C07320=1109.351,336.589,-83.150,-177.426,10.830,149.506
C07321=1109.354,336.377,-83.120,-177.429,10.829,149.507
C07322=1109.357,336.166,-83.091,-177.431,10.827,149.507
C07323=1109.361,335.954,-83.061,-177.435,10.824,149.507
C07324=1109.364,335.707,-83.027,-177.437,10.823,149.507
C07325=1109.368,335.458,-82.992,-177.440,10.820,149.507
C07326=1109.373,335.211,-82.959,-177.443,10.817,149.508
C07327=1109.376,334.963,-82.924,-177.447,10.815,149.508
C07328=1109.380,334.715,-82.890,-177.450,10.812,149.508
C07329=1109.385,334.468,-82.856,-177.453,10.810,149.508
C07330=1109.388,334.220,-82.822,-177.456,10.807,149.508
C07331=1109.393,333.973,-82.787,-177.460,10.805,149.509
C07332=1109.396,333.725,-82.753,-177.463,10.802,149.509
C07333=1109.400,333.478,-82.719,-177.466,10.799,149.509
C07334=1109.404,333.229,-82.685,-177.469,10.798,149.509
C07335=1109.408,332.982,-82.651,-177.472,10.795,149.509
C07336=1109.412,332.735,-82.617,-177.475,10.793,149.509
C07337=1109.416,332.487,-82.582,-177.478,10.790,149.510
C07338=1109.419,332.240,-82.549,-177.481,10.788,149.510
C07339=1109.424,331.991,-82.514,-177.484,10.785,149.510
C07340=1109.428,331.744,-82.481,-177.488,10.782,149.510
C07341=1109.431,331.497,-82.447,-177.491,10.780,149.510
C07342=1109.435,331.249,-82.412,-177.494,10.777,149.511
C07343=1109.440,331.001,-82.379,-177.497,10.776,149.511
C07344=1109.443,330.754,-82.345,-177.500,10.773,149.511
C07345=1109.447,330.506,-82.310,-177.503,10.771,149.511
C07346=1109.451,330.258,-82.277,-177.506,10.768,149.511
C07347=1109.455,330.011,-82.243,-177.510,10.765,149.512
C07348=1109.459,329.762,-82.209,-177.513,10.763,149.512
C07349=1109.463,329.515,-82.175,-177.516,10.760,149.512
C07350=1109.467,329.268,-82.141,-177.519,10.758,149.512
C07351=1109.471,329.019,-82.108,-177.522,10.755,149.512
C07352=1109.475,328.772,-82.074,-177.525,10.752,149.512
C07353=1109.479,328.524,-82.040,-177.528,10.751,149.513
C07354=1109.483,328.276,-82.006,-177.531,10.748,149.513
C07355=1109.487,328.029,-81.973,-177.534,10.746,149.513
C07356=1109.491,327.782,-81.939,-177.538,10.743,149.513
C07357=1109.496,327.534,-81.905,-177.541,10.741,149.513
C07358=1109.499,327.286,-81.871,-177.544,10.738,149.514
C07359=1109.503,327.038,-81.838,-177.547,10.735,149.514
C07360=1109.507,326.791,-81.804,-177.550,10.733,149.514
C07361=1109.510,326.543,-81.770,-177.553,10.730,149.514
C07362=1109.514,326.295,-81.736,-177.557,10.728,149.514
C07363=1109.519,326.047,-81.703,-177.559,10.726,149.515
C07364=1109.523,325.800,-81.669,-177.562,10.723,149.515
C07365=1109.526,325.552,-81.635,-177.566,10.721,149.515
C07366=1109.531,325.304,-81.602,-177.569,10.718,149.515
C07367=1109.534,325.057,-81.568,-177.572,10.716,149.515
C07368=1109.538,324.809,-81.535,-177.575,10.713,149.515
C07369=1109.543,324.562,-81.502,-177.579,10.711,149.516
C07370=1109.546,324.314,-81.468,-177.581,10.708,149.516
C07371=1109.550,324.066,-81.434,-177.585,10.706,149.516
C07372=1109.554,323.854,-81.406,-177.587,10.704,149.516
C07373=1109.557,323.642,-81.377,-177.590,10.702,149.516
C07374=1109.561,323.430,-81.348,-177.593,10.699,149.516
C07375=1109.564,323.219,-81.320,-177.595,10.697,149.517
C07376=1109.567,323.006,-81.291,-177.598,10.695,149.517
C07377=1109.571,322.794,-81.263,-177.601,10.693,149.517
C07378=1109.575,322.582,-81.234,-177.603,10.691,149.517
C07379=1109.577,322.370,-81.205,-177.606,10.689,149.517
C07380=1109.581,322.122,-81.172,-177.609,10.687,149.517
C07381=1109.586,321.874,-81.139,-177.612,10.684,149.518
C07382=1109.589,321.627,-81.105,-177.615,10.681,149.518
C07383=1109.594,321.379,-81.072,-177.618,10.679,149.518
C07384=1109.597,321.131,-81.039,-177.621,10.676,149.518
C07385=1109.601,320.883,-81.005,-177.625,10.674,149.518
C07386=1109.605,320.635,-80.972,-177.628,10.671,149.518
C07387=1109.609,320.388,-80.939,-177.630,10.669,149.519
C07388=1109.614,320.140,-80.906,-177.634,10.667,149.519
C07389=1109.618,319.892,-80.873,-177.637,10.664,149.519
C07390=1109.621,319.645,-80.840,-177.640,10.662,149.519
C07391=1109.625,319.397,-80.807,-177.643,10.659,149.519
C07392=1109.629,319.149,-80.773,-177.646,10.656,149.520
C07393=1109.633,318.902,-80.740,-177.649,10.654,149.520
C07394=1109.637,318.654,-80.707,-177.652,10.651,149.520
C07395=1109.641,318.406,-80.674,-177.656,10.649,149.520
C07396=1109.645,318.158,-80.641,-177.658,10.647,149.520
C07397=1109.650,317.910,-80.608,-177.661,10.644,149.520
C07398=1109.653,317.663,-80.575,-177.665,10.642,149.521
C07399=1109.657,317.415,-80.542,-177.668,10.639,149.521
C07400=1109.661,317.167,-80.509,-177.671,10.637,149.521
C07401=1109.665,316.919,-80.476,-177.674,10.634,149.521
C07402=1109.669,316.672,-80.443,-177.677,10.631,149.521
C07403=1109.672,316.424,-80.410,-177.681,10.629,149.522
C07404=1109.676,316.176,-80.377,-177.683,10.626,149.522
C07405=1109.681,315.928,-80.343,-177.687,10.624,149.522
C07406=1109.685,315.680,-80.311,-177.689,10.622,149.522
C07407=1109.689,315.432,-80.278,-177.692,10.619,149.522
C07408=1109.693,315.185,-80.245,-177.696,10.617,149.523
C07409=1109.697,314.937,-80.212,-177.699,10.614,149.523
C07410=1109.701,314.689,-80.179,-177.702,10.612,149.523
C07411=1109.705,314.441,-80.146,-177.705,10.609,149.523
C07412=1109.709,314.193,-80.114,-177.708,10.606,149.523
C07413=1109.713,313.946,-80.081,-177.711,10.604,149.523
C07414=1109.717,313.697,-80.048,-177.714,10.601,149.524
C07415=1109.721,313.450,-80.016,-177.717,10.600,149.524
C07416=1109.725,313.202,-79.983,-177.720,10.597,149.524
C07417=1109.729,312.954,-79.950,-177.723,10.594,149.524
C07418=1109.733,312.706,-79.918,-177.726,10.592,149.524
C07419=1109.737,312.459,-79.884,-177.730,10.589,149.524
C07420=1109.741,312.210,-79.852,-177.733,10.586,149.525
C07421=1109.745,311.964,-79.820,-177.736,10.584,149.525
C07422=1109.749,311.716,-79.787,-177.739,10.581,149.525
C07423=1109.754,311.468,-79.754,-177.742,10.579,149.525
C07424=1109.757,311.220,-79.722,-177.746,10.576,149.525
C07425=1109.762,310.972,-79.689,-177.748,10.574,149.525
C07426=1109.766,310.724,-79.656,-177.751,10.572,149.526
C07427=1109.769,310.476,-79.624,-177.754,10.569,149.526
C07428=1109.773,310.264,-79.596,-177.757,10.567,149.526
C07429=1109.776,310.052,-79.568,-177.760,10.565,149.526
C07430=1109.780,309.840,-79.540,-177.762,10.563,149.526
C07431=1109.783,309.627,-79.513,-177.765,10.560,149.527
C07432=1109.787,309.415,-79.484,-177.768,10.558,149.527
C07433=1109.790,309.203,-79.456,-177.770,10.556,149.527
C07434=1109.794,308.991,-79.429,-177.773,10.554,149.527
C07435=1109.797,308.779,-79.401,-177.776,10.552,149.527
C07436=1109.801,308.532,-79.369,-177.779,10.549,149.527
C07437=1109.805,308.283,-79.336,-177.782,10.546,149.527
C07438=1109.809,308.035,-79.304,-177.785,10.544,149.528
C07439=1109.814,307.788,-79.272,-177.787,10.542,149.528
C07440=1109.817,307.540,-79.240,-177.791,10.540,149.528
C07441=1109.822,307.292,-79.207,-177.794,10.537,149.528
C07442=1109.825,307.044,-79.175,-177.797,10.534,149.528
C07443=1109.830,306.796,-79.142,-177.800,10.532,149.528
C07444=1109.833,306.548,-79.111,-177.803,10.529,149.529
C07445=1109.838,306.301,-79.078,-177.806,10.526,149.529
C07446=1109.842,306.053,-79.046,-177.810,10.524,149.529
C07447=1109.846,305.804,-79.013,-177.812,10.521,149.529
C07448=1109.850,305.556,-78.982,-177.815,10.520,149.529
C07449=1109.854,305.309,-78.948,-177.818,10.517,149.529
C07450=1109.858,305.061,-78.917,-177.821,10.514,149.530
C07451=1109.862,304.813,-78.885,-177.824,10.512,149.530
C07452=1109.866,304.565,-78.853,-177.828,10.509,149.530
C07453=1109.870,304.317,-78.821,-177.831,10.506,149.530
C07454=1109.874,304.069,-78.788,-177.834,10.504,149.530
C07455=1109.879,303.822,-78.756,-177.837,10.502,149.531
C07456=1109.882,303.574,-78.724,-177.840,10.499,149.531
C07457=1109.887,303.325,-78.692,-177.843,10.497,149.531
C07458=1109.890,303.077,-78.660,-177.846,10.494,149.531
C07459=1109.895,302.830,-78.629,-177.849,10.492,149.531
C07460=1109.899,302.582,-78.596,-177.852,10.489,149.531
C07461=1109.903,302.334,-78.564,-177.855,10.487,149.532
C07462=1109.907,302.086,-78.533,-177.858,10.484,149.532
C07463=1109.912,301.838,-78.500,-177.862,10.482,149.532
C07464=1109.915,301.590,-78.469,-177.865,10.479,149.532
C07465=1109.919,301.342,-78.437,-177.868,10.476,149.532
C07466=1109.924,301.094,-78.405,-177.871,10.474,149.532
C07467=1109.928,300.846,-78.373,-177.874,10.472,149.533
C07468=1109.932,300.598,-78.341,-177.876,10.469,149.533
C07469=1109.936,300.351,-78.309,-177.880,10.467,149.533
C07470=1109.940,300.103,-78.277,-177.883,10.464,149.533
C07471=1109.944,299.854,-78.245,-177.886,10.461,149.533
C07472=1109.948,299.607,-78.214,-177.889,10.459,149.534
C07473=1109.952,299.359,-78.182,-177.892,10.456,149.534
C07474=1109.956,299.111,-78.150,-177.895,10.454,149.534
C07475=1109.961,298.863,-78.118,-177.899,10.451,149.534
C07476=1109.964,298.615,-78.086,-177.901,10.449,149.534
C07477=1109.968,298.367,-78.054,-177.904,10.447,149.535
C07478=1109.973,298.119,-78.023,-177.907,10.444,149.535
C07479=1109.976,297.871,-77.992,-177.910,10.441,149.535
C07480=1109.980,297.623,-77.960,-177.913,10.439,149.535
C07481=1109.985,297.376,-77.928,-177.916,10.436,149.535
C07482=1109.989,297.128,-77.896,-177.920,10.433,149.535
C07483=1109.993,296.879,-77.865,-177.923,10.431,149.535
C07484=1109.997,296.667,-77.838,-177.925,10.429,149.536
C07485=1110.000,296.455,-77.811,-177.928,10.427,149.536
C07486=1110.004,296.243,-77.784,-177.931,10.424,149.536
C07487=1110.008,296.030,-77.757,-177.933,10.422,149.536
C07488=1110.010,295.819,-77.730,-177.936,10.421,149.536
C07489=1110.014,295.606,-77.702,-177.939,10.418,149.536
C07490=1110.018,295.394,-77.675,-177.941,10.416,149.536
C07491=1110.021,295.181,-77.648,-177.943,10.414,149.537
C07492=1110.025,294.933,-77.618,-177.946,10.411,149.537
C07493=1110.029,294.685,-77.586,-177.949,10.409,149.537
C07494=1110.033,294.437,-77.555,-177.953,10.406,149.537
C07495=1110.037,294.189,-77.523,-177.956,10.404,149.537
C07496=1110.041,293.941,-77.491,-177.959,10.401,149.538
C07497=1110.046,293.693,-77.461,-177.962,10.398,149.538
C07498=1110.049,293.445,-77.429,-177.965,10.397,149.538
C07499=1110.054,293.197,-77.398,-177.968,10.394,149.538
C07500=1110.058,292.949,-77.366,-177.971,10.391,149.538
C07501=1110.062,292.701,-77.335,-177.974,10.389,149.538
C07502=1110.066,292.453,-77.304,-177.977,10.386,149.539
C07503=1110.070,292.205,-77.273,-177.980,10.384,149.539
C07504=1110.074,291.957,-77.241,-177.983,10.381,149.539
C07505=1110.078,291.709,-77.210,-177.986,10.378,149.539
C07506=1110.082,291.461,-77.178,-177.989,10.376,149.539
C07507=1110.087,291.213,-77.147,-177.992,10.374,149.539
C07508=1110.091,290.965,-77.116,-177.995,10.371,149.540
C07509=1110.095,290.717,-77.085,-177.998,10.369,149.540
C07510=1110.099,290.469,-77.053,-178.001,10.366,149.540
C07511=1110.102,290.221,-77.023,-178.005,10.364,149.540
C07512=1110.107,289.973,-76.992,-178.007,10.361,149.540
C07513=1110.111,289.726,-76.960,-178.010,10.358,149.540
C07514=1110.115,289.477,-76.929,-178.014,10.356,149.541
C07515=1110.120,289.229,-76.898,-178.016,10.354,149.541
C07516=1110.124,288.981,-76.867,-178.019,10.351,149.541
C07517=1110.128,288.733,-76.836,-178.022,10.348,149.541
C07518=1110.132,288.485,-76.805,-178.026,10.346,149.541
C07519=1110.136,288.237,-76.774,-178.029,10.343,149.541
C07520=1110.140,287.989,-76.743,-178.032,10.341,149.542
C07521=1110.144,287.741,-76.712,-178.035,10.338,149.542
C07522=1110.149,287.493,-76.681,-178.038,10.335,149.542
C07523=1110.152,287.245,-76.650,-178.041,10.334,149.542
C07524=1110.157,286.997,-76.619,-178.043,10.331,149.542
C07525=1110.161,286.749,-76.588,-178.047,10.328,149.543
C07526=1110.165,286.501,-76.557,-178.050,10.326,149.543
C07527=1110.169,286.252,-76.527,-178.053,10.323,149.543
C07528=1110.173,286.005,-76.495,-178.056,10.320,149.543
C07529=1110.177,285.757,-76.465,-178.059,10.318,149.543
C07530=1110.182,285.508,-76.433,-178.062,10.315,149.543
C07531=1110.185,285.261,-76.403,-178.065,10.313,149.544
C07532=1110.190,285.013,-76.372,-178.068,10.311,149.544
C07533=1110.194,284.764,-76.341,-178.071,10.308,149.544
C07534=1110.198,284.516,-76.311,-178.074,10.305,149.544
C07535=1110.202,284.268,-76.280,-178.077,10.303,149.544
C07536=1110.207,284.020,-76.249,-178.080,10.300,149.544
C07537=1110.210,283.772,-76.219,-178.083,10.298,149.545
C07538=1110.215,283.524,-76.188,-178.086,10.295,149.545
C07539=1110.219,283.275,-76.157,-178.090,10.293,149.545
C07540=1110.223,283.064,-76.131,-178.092,10.291,149.545
C07541=1110.226,282.851,-76.105,-178.094,10.289,149.545
C07542=1110.230,282.638,-76.079,-178.097,10.286,149.545
C07543=1110.233,282.426,-76.052,-178.100,10.284,149.545
C07544=1110.237,282.214,-76.026,-178.102,10.282,149.546
C07545=1110.241,282.001,-76.000,-178.105,10.280,149.546
C07546=1110.244,281.789,-75.973,-178.107,10.277,149.546
C07547=1110.247,281.577,-75.948,-178.110,10.275,149.546
C07548=1110.252,281.329,-75.917,-178.113,10.273,149.546
C07549=1110.255,281.080,-75.886,-178.116,10.270,149.546
C07550=1110.260,280.832,-75.856,-178.119,10.268,149.547
C07551=1110.264,280.585,-75.826,-178.122,10.265,149.547
C07552=1110.268,280.335,-75.795,-178.125,10.262,149.547
C07553=1110.272,280.088,-75.765,-178.129,10.260,149.547
C07554=1110.277,279.840,-75.734,-178.131,10.258,149.547
C07555=1110.281,279.592,-75.703,-178.134,10.255,149.547
C07556=1110.285,279.344,-75.673,-178.137,10.252,149.548
C07557=1110.289,279.095,-75.643,-178.140,10.250,149.548
C07558=1110.293,278.847,-75.613,-178.143,10.247,149.548
C07559=1110.298,278.599,-75.582,-178.146,10.244,149.548
C07560=1110.302,278.352,-75.552,-178.149,10.242,149.548
C07561=1110.305,278.103,-75.522,-178.152,10.239,149.548
C07562=1110.310,277.855,-75.491,-178.155,10.237,149.548
C07563=1110.314,277.607,-75.461,-178.158,10.234,149.549
C07564=1110.319,277.358,-75.431,-178.160,10.232,149.549
C07565=1110.323,277.111,-75.401,-178.164,10.229,149.549
C07566=1110.326,276.862,-75.370,-178.167,10.227,149.549
C07567=1110.331,276.614,-75.340,-178.170,10.224,149.549
C07568=1110.335,276.366,-75.310,-178.173,10.221,149.549
C07569=1110.339,276.118,-75.279,-178.176,10.218,149.549
C07570=1110.344,275.870,-75.250,-178.179,10.216,149.550
C07571=1110.347,275.622,-75.219,-178.182,10.213,149.550
C07572=1110.352,275.373,-75.189,-178.185,10.210,149.550
C07573=1110.356,275.125,-75.159,-178.187,10.208,149.550
C07574=1110.360,274.877,-75.130,-178.190,10.206,149.550
C07575=1110.364,274.629,-75.099,-178.193,10.203,149.550
C07576=1110.369,274.381,-75.069,-178.196,10.200,149.550
C07577=1110.372,274.133,-75.039,-178.199,10.197,149.550
C07578=1110.377,273.884,-75.009,-178.202,10.195,149.550
C07579=1110.381,273.636,-74.979,-178.205,10.192,149.551
C07580=1110.385,273.388,-74.949,-178.207,10.190,149.551
C07581=1110.389,273.140,-74.918,-178.210,10.187,149.551
C07582=1110.394,272.892,-74.889,-178.213,10.185,149.551
C07583=1110.397,272.644,-74.859,-178.216,10.182,149.551
C07584=1110.402,272.396,-74.829,-178.219,10.179,149.551
C07585=1110.407,272.147,-74.799,-178.222,10.176,149.551
C07586=1110.410,271.899,-74.769,-178.225,10.174,149.551
C07587=1110.414,271.651,-74.739,-178.227,10.172,149.552
C07588=1110.418,271.403,-74.709,-178.230,10.169,149.552
C07589=1110.422,271.155,-74.680,-178.233,10.166,149.552
C07590=1110.427,270.906,-74.650,-178.236,10.163,149.552
C07591=1110.431,270.659,-74.619,-178.239,10.161,149.552
C07592=1110.435,270.410,-74.590,-178.242,10.158,149.552
C07593=1110.439,270.162,-74.561,-178.244,10.156,149.552
C07594=1110.443,269.914,-74.531,-178.247,10.153,149.552
C07595=1110.448,269.666,-74.500,-178.250,10.150,149.552
C07596=1110.452,269.452,-74.475,-178.253,10.148,149.552
C07597=1110.455,269.241,-74.450,-178.255,10.146,149.553
C07598=1110.459,269.029,-74.425,-178.258,10.144,149.553
C07599=1110.462,268.815,-74.400,-178.260,10.142,149.553
C07600=1110.466,268.603,-74.374,-178.262,10.140,149.553
C07601=1110.469,268.390,-74.348,-178.265,10.138,149.553
C07602=1110.473,268.178,-74.323,-178.268,10.135,149.553
C07603=1110.477,267.965,-74.297,-178.270,10.133,149.553
C07604=1110.481,267.717,-74.268,-178.273,10.130,149.553
C07605=1110.485,267.468,-74.238,-178.275,10.128,149.554
C07606=1110.489,267.221,-74.208,-178.278,10.125,149.554
C07607=1110.493,266.972,-74.179,-178.281,10.123,149.554
C07608=1110.497,266.724,-74.149,-178.284,10.120,149.554
C07609=1110.501,266.476,-74.120,-178.286,10.118,149.554
C07610=1110.506,266.228,-74.090,-178.289,10.115,149.554
C07611=1110.510,265.980,-74.061,-178.292,10.112,149.554
C07612=1110.515,265.732,-74.032,-178.295,10.110,149.554
C07613=1110.520,265.483,-74.002,-178.297,10.108,149.554
C07614=1110.524,265.235,-73.972,-178.300,10.105,149.554
C07615=1110.528,264.987,-73.943,-178.303,10.102,149.555
C07616=1110.532,264.738,-73.914,-178.306,10.100,149.555
C07617=1110.536,264.490,-73.884,-178.309,10.098,149.555
C07618=1110.540,264.242,-73.855,-178.312,10.095,149.555
C07619=1110.545,263.994,-73.825,-178.315,10.092,149.555
C07620=1110.549,263.745,-73.796,-178.318,10.089,149.555
C07621=1110.552,263.497,-73.767,-178.321,10.087,149.555
C07622=1110.556,263.249,-73.737,-178.324,10.084,149.556
C07623=1110.561,263.001,-73.708,-178.327,10.082,149.556
C07624=1110.565,262.753,-73.679,-178.330,10.079,149.556
C07625=1110.570,262.504,-73.650,-178.333,10.076,149.556
C07626=1110.574,262.256,-73.621,-178.336,10.073,149.556
C07627=1110.578,262.008,-73.591,-178.339,10.071,149.556
C07628=1110.582,261.760,-73.562,-178.342,10.068,149.556
C07629=1110.587,261.511,-73.532,-178.345,10.065,149.556
C07630=1110.591,261.263,-73.503,-178.347,10.063,149.557
C07631=1110.596,261.015,-73.475,-178.350,10.060,149.557
C07632=1110.600,260.767,-73.445,-178.353,10.058,149.557
C07633=1110.603,260.519,-73.416,-178.356,10.055,149.557
C07634=1110.608,260.270,-73.387,-178.359,10.052,149.557
C07635=1110.612,260.021,-73.358,-178.362,10.049,149.557
C07636=1110.616,259.773,-73.329,-178.364,10.046,149.557
C07637=1110.621,259.525,-73.299,-178.367,10.043,149.557
C07638=1110.625,259.277,-73.271,-178.370,10.041,149.557
C07639=1110.629,259.029,-73.242,-178.373,10.038,149.557
C07640=1110.633,258.780,-73.212,-178.376,10.035,149.557
C07641=1110.638,258.532,-73.184,-178.379,10.032,149.558
C07642=1110.642,258.283,-73.154,-178.381,10.030,149.557
C07643=1110.646,258.036,-73.126,-178.384,10.027,149.558
C07644=1110.650,257.787,-73.097,-178.387,10.024,149.558
C07645=1110.655,257.539,-73.068,-178.390,10.022,149.558
C07646=1110.659,257.291,-73.038,-178.392,10.019,149.558
C07647=1110.663,257.043,-73.010,-178.395,10.016,149.558
C07648=1110.667,256.794,-72.981,-178.398,10.013,149.558
C07649=1110.672,256.546,-72.952,-178.401,10.010,149.558
C07650=1110.675,256.298,-72.923,-178.403,10.007,149.558
C07651=1110.680,256.049,-72.895,-178.406,10.005,149.558
C07652=1110.684,255.836,-72.870,-178.408,10.003,149.558
C07653=1110.687,255.624,-72.845,-178.410,10.001,149.558
C07654=1110.691,255.412,-72.820,-178.412,9.999,149.558
C07655=1110.694,255.198,-72.795,-178.413,9.997,149.558
C07656=1110.698,254.986,-72.771,-178.415,9.995,149.558
C07657=1110.702,254.773,-72.746,-178.417,9.993,149.558
C07658=1110.706,254.561,-72.722,-178.420,9.991,149.558
C07659=1110.709,254.348,-72.697,-178.421,9.990,149.558
C07660=1110.714,254.099,-72.669,-178.424,9.986,149.558
C07661=1110.718,253.851,-72.639,-178.426,9.984,149.558
C07662=1110.722,253.603,-72.611,-178.429,9.982,149.559
C07663=1110.727,253.354,-72.583,-178.431,9.980,149.559
C07664=1110.730,253.106,-72.554,-178.434,9.977,149.559
C07665=1110.735,252.857,-72.525,-178.437,9.975,149.559
C07666=1110.740,252.609,-72.497,-178.440,9.973,149.559
C07667=1110.743,252.361,-72.468,-178.442,9.971,149.559
C07668=1110.748,252.112,-72.439,-178.445,9.968,149.559
C07669=1110.752,251.865,-72.411,-178.448,9.965,149.560
C07670=1110.756,251.616,-72.382,-178.452,9.963,149.560
C07671=1110.760,251.368,-72.354,-178.454,9.961,149.560
C07672=1110.765,251.120,-72.325,-178.457,9.958,149.560
C07673=1110.769,250.871,-72.296,-178.460,9.956,149.560
C07674=1110.773,250.623,-72.268,-178.463,9.953,149.561
C07675=1110.778,250.375,-72.239,-178.466,9.950,149.561
C07676=1110.782,250.126,-72.211,-178.469,9.948,149.561
C07677=1110.786,249.878,-72.182,-178.473,9.944,149.561
C07678=1110.790,249.630,-72.154,-178.476,9.941,149.561
C07679=1110.795,249.381,-72.125,-178.479,9.939,149.561
C07680=1110.799,249.133,-72.097,-178.483,9.935,149.562
C07681=1110.803,248.884,-72.069,-178.486,9.933,149.562
C07682=1110.807,248.636,-72.041,-178.489,9.930,149.562
C07683=1110.811,248.388,-72.012,-178.492,9.926,149.562
C07684=1110.816,248.139,-71.983,-178.496,9.923,149.562
C07685=1110.820,247.892,-71.956,-178.499,9.920,149.562
C07686=1110.825,247.643,-71.927,-178.502,9.917,149.562
C07687=1110.829,247.395,-71.899,-178.505,9.914,149.562
C07688=1110.833,247.146,-71.871,-178.508,9.911,149.562
C07689=1110.837,246.897,-71.842,-178.510,9.908,149.562
C07690=1110.842,246.649,-71.814,-178.512,9.905,149.562
C07691=1110.846,246.401,-71.786,-178.515,9.902,149.562
C07692=1110.851,246.153,-71.758,-178.517,9.900,149.562
C07693=1110.854,245.904,-71.730,-178.520,9.897,149.562
C07694=1110.859,245.656,-71.701,-178.522,9.895,149.562
C07695=1110.863,245.407,-71.673,-178.524,9.892,149.562
C07696=1110.867,245.159,-71.645,-178.527,9.889,149.562
C07697=1110.872,244.911,-71.617,-178.529,9.887,149.562
C07698=1110.876,244.663,-71.589,-178.531,9.883,149.562
C07699=1110.880,244.414,-71.561,-178.534,9.881,149.562
C07700=1110.885,244.165,-71.533,-178.536,9.878,149.562
C07701=1110.889,243.917,-71.505,-178.539,9.876,149.562
C07702=1110.894,243.669,-71.477,-178.541,9.873,149.562
C07703=1110.897,243.420,-71.449,-178.544,9.871,149.562
C07704=1110.902,243.172,-71.421,-178.546,9.868,149.562
C07705=1110.906,242.924,-71.393,-178.549,9.865,149.562
C07706=1110.911,242.676,-71.365,-178.551,9.863,149.562
C07707=1110.915,242.426,-71.337,-178.554,9.860,149.562
C07708=1110.918,242.214,-71.313,-178.556,9.858,149.562
C07709=1110.922,242.001,-71.289,-178.558,9.856,149.562
C07710=1110.926,241.788,-71.265,-178.560,9.854,149.562
C07711=1110.930,241.575,-71.241,-178.562,9.852,149.562
C07712=1110.933,241.363,-71.217,-178.564,9.849,149.562
C07713=1110.937,241.150,-71.194,-178.567,9.847,149.562
C07714=1110.941,240.937,-71.170,-178.569,9.844,149.562
C07715=1110.944,240.724,-71.146,-178.571,9.842,149.563
C07716=1110.949,240.476,-71.118,-178.573,9.840,149.563
C07717=1110.953,240.227,-71.090,-178.576,9.837,149.563
C07718=1110.957,239.979,-71.062,-178.579,9.835,149.563
C07719=1110.961,239.731,-71.034,-178.581,9.833,149.563
C07720=1110.966,239.482,-71.007,-178.584,9.829,149.563
C07721=1110.970,239.234,-70.979,-178.587,9.827,149.563
C07722=1110.975,238.985,-70.951,-178.589,9.825,149.563
C07723=1110.979,238.737,-70.923,-178.592,9.822,149.563
C07724=1110.983,238.488,-70.895,-178.594,9.820,149.563
C07725=1110.988,238.240,-70.868,-178.597,9.817,149.563
C07726=1110.992,237.992,-70.840,-178.600,9.814,149.563
C07727=1110.996,237.743,-70.813,-178.603,9.811,149.563
C07728=1111.001,237.495,-70.785,-178.605,9.809,149.564
C07729=1111.004,237.246,-70.757,-178.608,9.806,149.564
C07730=1111.009,236.998,-70.730,-178.610,9.804,149.564
C07731=1111.013,236.750,-70.702,-178.613,9.802,149.564
C07732=1111.017,236.501,-70.675,-178.616,9.799,149.564
C07733=1111.022,236.253,-70.647,-178.619,9.796,149.564
C07734=1111.027,236.004,-70.619,-178.621,9.794,149.564
C07735=1111.031,235.755,-70.591,-178.624,9.791,149.564
C07736=1111.035,235.507,-70.564,-178.626,9.788,149.564
C07737=1111.040,235.259,-70.536,-178.629,9.785,149.564
C07738=1111.044,235.010,-70.509,-178.632,9.783,149.564
C07739=1111.049,234.761,-70.482,-178.634,9.780,149.564
C07740=1111.053,234.514,-70.454,-178.637,9.778,149.565
C07741=1111.057,234.264,-70.427,-178.640,9.775,149.565
C07742=1111.061,234.017,-70.400,-178.643,9.772,149.565
C07743=1111.065,233.768,-70.373,-178.645,9.770,149.565
C07744=1111.070,233.520,-70.345,-178.648,9.767,149.565
C07745=1111.074,233.271,-70.317,-178.651,9.764,149.565
C07746=1111.078,233.023,-70.290,-178.654,9.762,149.565
C07747=1111.083,232.774,-70.263,-178.656,9.758,149.565
C07748=1111.087,232.526,-70.235,-178.659,9.756,149.565
C07749=1111.091,232.277,-70.208,-178.662,9.753,149.565
C07750=1111.096,232.029,-70.181,-178.665,9.751,149.565
C07751=1111.100,231.781,-70.153,-178.667,9.748,149.565
C07752=1111.104,231.532,-70.126,-178.670,9.745,149.565
C07753=1111.109,231.283,-70.099,-178.673,9.742,149.566
C07754=1111.113,231.035,-70.072,-178.676,9.739,149.566
C07755=1111.118,230.786,-70.045,-178.678,9.737,149.566
C07756=1111.122,230.539,-70.017,-178.681,9.733,149.566
C07757=1111.126,230.289,-69.990,-178.684,9.731,149.566
C07758=1111.131,230.041,-69.963,-178.687,9.728,149.566
C07759=1111.135,229.792,-69.936,-178.689,9.725,149.566
C07760=1111.139,229.544,-69.909,-178.692,9.722,149.566
C07761=1111.144,229.296,-69.882,-178.695,9.719,149.566
C07762=1111.148,229.047,-69.854,-178.698,9.716,149.566
C07763=1111.152,228.799,-69.827,-178.700,9.713,149.566
C07764=1111.156,228.586,-69.804,-178.703,9.710,149.566
C07765=1111.160,228.373,-69.782,-178.705,9.708,149.566
C07766=1111.164,228.160,-69.758,-178.708,9.705,149.566
C07767=1111.167,227.947,-69.735,-178.710,9.703,149.566
C07768=1111.171,227.734,-69.711,-178.712,9.701,149.566
C07769=1111.174,227.521,-69.689,-178.714,9.697,149.566
C07770=1111.178,227.308,-69.666,-178.716,9.695,149.566
C07771=1111.183,227.095,-69.642,-178.719,9.692,149.566
C07772=1111.187,226.846,-69.615,-178.722,9.689,149.566
C07773=1111.190,226.598,-69.589,-178.724,9.686,149.566
C07774=1111.195,226.349,-69.561,-178.727,9.683,149.566
C07775=1111.200,226.101,-69.534,-178.730,9.680,149.566
C07776=1111.204,225.853,-69.508,-178.732,9.677,149.566
C07777=1111.208,225.604,-69.481,-178.735,9.674,149.566
C07778=1111.213,225.356,-69.454,-178.737,9.671,149.566
C07779=1111.217,225.107,-69.427,-178.740,9.668,149.566
C07780=1111.222,224.859,-69.400,-178.742,9.665,149.566
C07781=1111.226,224.609,-69.374,-178.745,9.662,149.565
C07782=1111.230,224.361,-69.347,-178.747,9.659,149.565
C07783=1111.235,224.112,-69.320,-178.749,9.656,149.565
C07784=1111.239,223.864,-69.293,-178.752,9.653,149.565
C07785=1111.243,223.616,-69.266,-178.754,9.650,149.565
C07786=1111.248,223.367,-69.239,-178.757,9.647,149.565
C07787=1111.252,223.119,-69.214,-178.759,9.644,149.565
C07788=1111.257,222.870,-69.187,-178.762,9.641,149.565
C07789=1111.261,222.622,-69.160,-178.765,9.638,149.565
C07790=1111.265,222.373,-69.133,-178.767,9.634,149.565
C07791=1111.270,222.125,-69.106,-178.770,9.631,149.565
C07792=1111.274,221.876,-69.080,-178.772,9.628,149.565
C07793=1111.279,221.628,-69.053,-178.775,9.625,149.565
C07794=1111.283,221.379,-69.027,-178.777,9.622,149.565
C07795=1111.288,221.130,-69.000,-178.780,9.619,149.565
C07796=1111.292,220.882,-68.974,-178.781,9.616,149.564
C07797=1111.296,220.634,-68.947,-178.784,9.613,149.564
C07798=1111.300,220.385,-68.921,-178.786,9.610,149.564
C07799=1111.305,220.136,-68.894,-178.789,9.607,149.564
C07800=1111.309,219.888,-68.868,-178.791,9.604,149.564
C07801=1111.314,219.639,-68.841,-178.794,9.601,149.564
C07802=1111.318,219.391,-68.815,-178.796,9.597,149.564
C07803=1111.323,219.142,-68.788,-178.798,9.595,149.564
C07804=1111.327,218.893,-68.762,-178.800,9.592,149.564
C07805=1111.331,218.645,-68.735,-178.803,9.589,149.564
C07806=1111.336,218.396,-68.709,-178.805,9.585,149.563
C07807=1111.340,218.148,-68.683,-178.807,9.582,149.563
C07808=1111.345,217.899,-68.656,-178.810,9.579,149.563
C07809=1111.348,217.651,-68.630,-178.812,9.577,149.563
C07810=1111.353,217.402,-68.604,-178.814,9.573,149.563
C07811=1111.357,217.153,-68.577,-178.817,9.570,149.563
C07812=1111.362,216.905,-68.551,-178.819,9.567,149.563
C07813=1111.366,216.656,-68.524,-178.821,9.565,149.563
C07814=1111.370,216.407,-68.499,-178.823,9.561,149.563
C07815=1111.374,216.159,-68.472,-178.826,9.558,149.562
C07816=1111.379,215.910,-68.446,-178.828,9.555,149.562
C07817=1111.383,215.662,-68.419,-178.830,9.553,149.562
C07818=1111.388,215.414,-68.394,-178.832,9.549,149.562
C07819=1111.393,215.165,-68.367,-178.835,9.546,149.562
C07820=1111.396,214.952,-68.345,-178.836,9.544,149.562
C07821=1111.400,214.738,-68.322,-178.838,9.541,149.562
C07822=1111.404,214.526,-68.300,-178.840,9.539,149.562
C07823=1111.407,214.312,-68.278,-178.842,9.537,149.562
C07824=1111.412,214.099,-68.255,-178.844,9.534,149.562
C07825=1111.415,213.887,-68.232,-178.846,9.532,149.561
C07826=1111.418,213.673,-68.210,-178.848,9.528,149.561
C07827=1111.423,213.460,-68.188,-178.850,9.526,149.561
C07828=1111.427,213.212,-68.162,-178.852,9.523,149.561
C07829=1111.431,212.963,-68.136,-178.855,9.520,149.561
C07830=1111.436,212.714,-68.109,-178.859,9.516,149.561
C07831=1111.440,212.465,-68.084,-178.861,9.513,149.561
C07832=1111.445,212.217,-68.058,-178.864,9.511,149.561
C07833=1111.449,211.969,-68.032,-178.867,9.507,149.561
C07834=1111.453,211.720,-68.006,-178.870,9.504,149.561
C07835=1111.458,211.471,-67.980,-178.873,9.501,149.561
C07836=1111.462,211.222,-67.954,-178.876,9.498,149.561
C07837=1111.467,210.974,-67.928,-178.879,9.494,149.561
C07838=1111.471,210.726,-67.902,-178.882,9.491,149.562
C07839=1111.475,210.477,-67.876,-178.884,9.488,149.561
C07840=1111.480,210.228,-67.850,-178.887,9.486,149.562
C07841=1111.485,209.979,-67.824,-178.890,9.483,149.562
C07842=1111.489,209.731,-67.798,-178.893,9.479,149.562
C07843=1111.494,209.483,-67.773,-178.896,9.476,149.562
C07844=1111.498,209.234,-67.747,-178.899,9.473,149.562
C07845=1111.502,208.985,-67.721,-178.902,9.470,149.562
C07846=1111.506,208.736,-67.696,-178.905,9.468,149.562
C07847=1111.511,208.488,-67.670,-178.907,9.464,149.562
C07848=1111.516,208.239,-67.644,-178.910,9.462,149.562
C07849=1111.520,207.990,-67.618,-178.914,9.458,149.562
C07850=1111.524,207.741,-67.592,-178.917,9.455,149.562
C07851=1111.529,207.493,-67.567,-178.919,9.452,149.562
C07852=1111.534,207.244,-67.541,-178.922,9.450,149.562
C07853=1111.538,206.996,-67.516,-178.925,9.447,149.563
C07854=1111.543,206.747,-67.490,-178.928,9.444,149.563
C07855=1111.547,206.499,-67.464,-178.931,9.441,149.563
C07856=1111.551,206.250,-67.439,-178.934,9.438,149.563
C07857=1111.556,206.002,-67.413,-178.936,9.435,149.563
C07858=1111.560,205.753,-67.388,-178.939,9.432,149.563
C07859=1111.564,205.504,-67.362,-178.942,9.430,149.563
C07860=1111.569,205.256,-67.336,-178.946,9.426,149.563
C07861=1111.574,205.007,-67.311,-178.948,9.423,149.563
C07862=1111.578,204.758,-67.286,-178.951,9.420,149.563
C07863=1111.583,204.510,-67.260,-178.954,9.418,149.563
C07864=1111.587,204.261,-67.235,-178.957,9.415,149.564
C07865=1111.591,204.012,-67.209,-178.960,9.412,149.564
C07866=1111.596,203.764,-67.183,-178.962,9.409,149.564
C07867=1111.601,203.515,-67.158,-178.965,9.406,149.564
C07868=1111.604,203.266,-67.133,-178.968,9.403,149.564
C07869=1111.609,203.018,-67.108,-178.971,9.400,149.564
C07870=1111.613,202.769,-67.083,-178.974,9.398,149.564
C07871=1111.618,202.520,-67.057,-178.977,9.395,149.564
C07872=1111.622,202.272,-67.032,-178.979,9.392,149.564
C07873=1111.627,202.023,-67.006,-178.982,9.389,149.564
C07874=1111.632,201.774,-66.981,-178.985,9.386,149.564
C07875=1111.635,201.526,-66.956,-178.988,9.383,149.564
C07876=1111.639,201.312,-66.935,-178.991,9.380,149.564
C07877=1111.643,201.099,-66.913,-178.992,9.378,149.564
C07878=1111.647,200.886,-66.892,-178.995,9.375,149.565
C07879=1111.651,200.673,-66.870,-178.997,9.373,149.565
C07880=1111.654,200.459,-66.848,-179.000,9.371,149.565
C07881=1111.658,200.247,-66.827,-179.002,9.368,149.565
C07882=1111.662,200.033,-66.805,-179.004,9.366,149.565
C07883=1111.666,199.820,-66.783,-179.007,9.363,149.565
C07884=1111.671,199.571,-66.759,-179.010,9.360,149.565
C07885=1111.675,199.322,-66.733,-179.012,9.357,149.565
C07886=1111.680,199.073,-66.708,-179.015,9.354,149.565
C07887=1111.684,198.825,-66.683,-179.018,9.351,149.565
C07888=1111.688,198.576,-66.657,-179.020,9.348,149.565
C07889=1111.693,198.328,-66.633,-179.023,9.345,149.565
C07890=1111.698,198.078,-66.608,-179.026,9.342,149.565
C07891=1111.702,197.831,-66.583,-179.028,9.339,149.565
C07892=1111.706,197.581,-66.558,-179.031,9.336,149.565
C07893=1111.711,197.333,-66.532,-179.034,9.333,149.565
C07894=1111.715,197.084,-66.508,-179.037,9.329,149.565
C07895=1111.720,196.836,-66.482,-179.040,9.326,149.565
C07896=1111.724,196.586,-66.457,-179.042,9.323,149.565
C07897=1111.729,196.338,-66.433,-179.045,9.320,149.565
C07898=1111.733,196.089,-66.408,-179.046,9.317,149.565
C07899=1111.738,195.840,-66.383,-179.049,9.314,149.565
C07900=1111.742,195.592,-66.359,-179.051,9.312,149.564
C07901=1111.747,195.343,-66.333,-179.053,9.308,149.564
C07902=1111.751,195.095,-66.309,-179.055,9.306,149.564
C07903=1111.756,194.845,-66.284,-179.057,9.303,149.564
C07904=1111.760,194.597,-66.259,-179.059,9.301,149.564
C07905=1111.764,194.348,-66.234,-179.061,9.297,149.564
C07906=1111.769,194.099,-66.210,-179.063,9.295,149.564
C07907=1111.773,193.850,-66.185,-179.066,9.292,149.564
C07908=1111.778,193.602,-66.160,-179.067,9.289,149.564
C07909=1111.783,193.353,-66.135,-179.070,9.286,149.564
C07910=1111.787,193.104,-66.111,-179.071,9.284,149.563
C07911=1111.792,192.856,-66.086,-179.074,9.280,149.563
C07912=1111.796,192.607,-66.061,-179.076,9.278,149.563
C07913=1111.801,192.358,-66.036,-179.078,9.275,149.563
C07914=1111.805,192.110,-66.012,-179.080,9.273,149.563
C07915=1111.810,191.861,-65.987,-179.083,9.270,149.563
C07916=1111.814,191.612,-65.963,-179.085,9.267,149.563
C07917=1111.819,191.363,-65.938,-179.087,9.264,149.563
C07918=1111.823,191.115,-65.913,-179.089,9.262,149.563
C07919=1111.828,190.866,-65.888,-179.092,9.259,149.563
C07920=1111.832,190.617,-65.864,-179.094,9.255,149.563
C07921=1111.837,190.368,-65.839,-179.096,9.253,149.563
C07922=1111.841,190.120,-65.815,-179.098,9.250,149.563
C07923=1111.846,189.871,-65.790,-179.100,9.247,149.563
C07924=1111.850,189.622,-65.766,-179.103,9.244,149.563
C07925=1111.855,189.373,-65.741,-179.104,9.242,149.563
C07926=1111.859,189.124,-65.717,-179.107,9.239,149.562
C07927=1111.864,188.876,-65.692,-179.109,9.236,149.562
C07928=1111.868,188.627,-65.668,-179.111,9.233,149.562
C07929=1111.872,188.378,-65.644,-179.114,9.230,149.562
C07930=1111.877,188.129,-65.619,-179.116,9.227,149.562
C07931=1111.882,187.881,-65.595,-179.118,9.225,149.562
C07932=1111.886,187.668,-65.574,-179.120,9.223,149.562
C07933=1111.890,187.454,-65.552,-179.122,9.220,149.562
C07934=1111.893,187.241,-65.532,-179.125,9.217,149.562
C07935=1111.897,187.028,-65.511,-179.127,9.215,149.562
C07936=1111.901,186.815,-65.490,-179.129,9.213,149.562
C07937=1111.905,186.601,-65.469,-179.131,9.210,149.562
C07938=1111.909,186.388,-65.448,-179.133,9.208,149.562
C07939=1111.912,186.174,-65.428,-179.134,9.206,149.562
C07940=1111.917,185.925,-65.403,-179.137,9.203,149.562
C07941=1111.922,185.677,-65.379,-179.140,9.200,149.562
C07942=1111.926,185.428,-65.355,-179.141,9.197,149.562
C07943=1111.931,185.179,-65.330,-179.144,9.194,149.562
C07944=1111.935,184.930,-65.306,-179.146,9.191,149.562
C07945=1111.940,184.682,-65.282,-179.148,9.189,149.562
C07946=1111.945,184.433,-65.258,-179.151,9.186,149.562
C07947=1111.949,184.184,-65.234,-179.153,9.182,149.562
C07948=1111.953,183.935,-65.209,-179.156,9.179,149.562
C07949=1111.958,183.687,-65.185,-179.158,9.176,149.562
C07950=1111.963,183.438,-65.161,-179.160,9.174,149.562
C07951=1111.967,183.189,-65.137,-179.163,9.171,149.562
C07952=1111.971,182.940,-65.113,-179.165,9.168,149.562
C07953=1111.976,182.691,-65.089,-179.168,9.165,149.562
C07954=1111.981,182.443,-65.064,-179.170,9.162,149.562
C07955=1111.985,182.194,-65.041,-179.172,9.159,149.561
C07956=1111.990,181.945,-65.017,-179.175,9.156,149.561
C07957=1111.994,181.696,-64.992,-179.177,9.153,149.561
C07958=1111.998,181.447,-64.969,-179.180,9.150,149.561
C07959=1112.003,181.198,-64.944,-179.182,9.147,149.561
C07960=1112.008,180.950,-64.920,-179.185,9.144,149.561
C07961=1112.013,180.701,-64.897,-179.187,9.141,149.561
C07962=1112.016,180.452,-64.872,-179.189,9.138,149.561
C07963=1112.021,180.203,-64.849,-179.192,9.135,149.561
C07964=1112.025,179.954,-64.825,-179.194,9.132,149.561
C07965=1112.030,179.706,-64.801,-179.196,9.128,149.561
C07966=1112.035,179.457,-64.778,-179.199,9.125,149.561
C07967=1112.040,179.208,-64.753,-179.202,9.122,149.561
C07968=1112.044,178.959,-64.730,-179.204,9.119,149.561
C07969=1112.048,178.710,-64.705,-179.206,9.116,149.560
C07970=1112.053,178.461,-64.682,-179.208,9.113,149.560
C07971=1112.057,178.213,-64.658,-179.210,9.111,149.560
C07972=1112.062,177.964,-64.634,-179.212,9.108,149.560
C07973=1112.066,177.715,-64.610,-179.215,9.104,149.560
C07974=1112.071,177.466,-64.587,-179.216,9.102,149.560
C07975=1112.075,177.218,-64.563,-179.219,9.099,149.560
C07976=1112.080,176.969,-64.539,-179.221,9.095,149.560
C07977=1112.085,176.720,-64.515,-179.223,9.093,149.560
C07978=1112.089,176.471,-64.492,-179.225,9.090,149.560
C07979=1112.093,176.222,-64.468,-179.228,9.087,149.559
C07980=1112.098,175.973,-64.444,-179.229,9.084,149.559
C07981=1112.102,175.724,-64.421,-179.232,9.081,149.559
C07982=1112.107,175.476,-64.397,-179.234,9.078,149.559
C07983=1112.112,175.227,-64.373,-179.236,9.075,149.559
C07984=1112.116,174.978,-64.350,-179.238,9.072,149.559
C07985=1112.121,174.729,-64.326,-179.241,9.069,149.559
C07986=1112.125,174.480,-64.303,-179.242,9.066,149.559
C07987=1112.130,174.231,-64.279,-179.245,9.063,149.559
C07988=1112.133,174.018,-64.259,-179.246,9.061,149.559
C07989=1112.138,173.804,-64.238,-179.248,9.058,149.558
C07990=1112.142,173.591,-64.219,-179.250,9.056,149.558
C07991=1112.145,173.378,-64.198,-179.253,9.053,149.558
C07992=1112.150,173.164,-64.178,-179.254,9.050,149.558
C07993=1112.154,172.950,-64.158,-179.256,9.048,149.558
C07994=1112.157,172.738,-64.137,-179.258,9.045,149.558
C07995=1112.161,172.524,-64.117,-179.259,9.043,149.558
C07996=1112.165,172.275,-64.094,-179.262,9.040,149.558
C07997=1112.170,172.026,-64.071,-179.264,9.036,149.558
C07998=1112.175,171.777,-64.047,-179.266,9.034,149.558
C07999=1112.179,171.528,-64.023,-179.268,9.031,149.558
C08000=1112.184,171.279,-64.000,-179.271,9.028,149.557
C08001=1112.189,171.031,-63.977,-179.273,9.025,149.557
C08002=1112.193,170.782,-63.954,-179.275,9.022,149.557
C08003=1112.198,170.533,-63.931,-179.277,9.019,149.557
C08004=1112.202,170.285,-63.907,-179.279,9.016,149.557
C08005=1112.207,170.036,-63.883,-179.281,9.013,149.557
C08006=1112.212,169.787,-63.860,-179.284,9.010,149.557
C08007=1112.216,169.538,-63.837,-179.285,9.007,149.557
C08008=1112.220,169.289,-63.814,-179.288,9.004,149.557
C08009=1112.225,169.040,-63.791,-179.290,9.001,149.557
C08010=1112.230,168.791,-63.767,-179.293,8.997,149.556
C08011=1112.234,168.542,-63.744,-179.294,8.995,149.556
C08012=1112.239,168.293,-63.721,-179.297,8.992,149.556
C08013=1112.243,168.044,-63.698,-179.299,8.988,149.556
C08014=1112.248,167.795,-63.674,-179.302,8.985,149.556
C08015=1112.253,167.547,-63.651,-179.303,8.983,149.556
C08016=1112.258,167.298,-63.628,-179.306,8.979,149.556
C08017=1112.262,167.049,-63.605,-179.308,8.976,149.556
C08018=1112.267,166.800,-63.582,-179.310,8.974,149.556
C08019=1112.271,166.551,-63.559,-179.312,8.971,149.555
C08020=1112.276,166.302,-63.535,-179.315,8.967,149.555
C08021=1112.280,166.053,-63.512,-179.317,8.964,149.555
C08022=1112.285,165.804,-63.489,-179.319,8.962,149.555
C08023=1112.290,165.556,-63.466,-179.321,8.958,149.555
C08024=1112.294,165.307,-63.443,-179.323,8.955,149.555
C08025=1112.299,165.058,-63.420,-179.326,8.952,149.555
C08026=1112.303,164.809,-63.397,-179.327,8.949,149.555
C08027=1112.307,164.560,-63.375,-179.330,8.946,149.554
C08028=1112.312,164.311,-63.351,-179.332,8.943,149.554
C08029=1112.317,164.062,-63.328,-179.334,8.939,149.554
C08030=1112.321,163.814,-63.305,-179.337,8.936,149.554
C08031=1112.326,163.565,-63.282,-179.338,8.934,149.554
C08032=1112.330,163.316,-63.259,-179.341,8.931,149.554
C08033=1112.335,163.066,-63.237,-179.343,8.927,149.554
C08034=1112.340,162.817,-63.213,-179.345,8.924,149.554
C08035=1112.344,162.569,-63.191,-179.347,8.921,149.553
C08036=1112.349,162.320,-63.168,-179.349,8.918,149.553
C08037=1112.353,162.071,-63.146,-179.351,8.915,149.553
C08038=1112.358,161.822,-63.122,-179.354,8.912,149.553
C08039=1112.363,161.573,-63.099,-179.356,8.908,149.553
C08040=1112.367,161.325,-63.076,-179.358,8.906,149.553
C08041=1112.372,161.075,-63.054,-179.360,8.902,149.553
C08042=1112.376,160.826,-63.031,-179.363,8.899,149.553
C08043=1112.381,160.577,-63.008,-179.365,8.896,149.552
C08044=1112.386,160.364,-62.989,-179.367,8.893,149.552
C08045=1112.389,160.151,-62.970,-179.368,8.891,149.552
C08046=1112.392,159.937,-62.950,-179.371,8.888,149.552
C08047=1112.396,159.724,-62.930,-179.372,8.885,149.552
C08048=1112.401,159.510,-62.911,-179.374,8.882,149.552
C08049=1112.405,159.297,-62.892,-179.376,8.879,149.552
C08050=1112.408,159.083,-62.872,-179.378,8.877,149.551
C08051=1112.413,158.869,-62.853,-179.380,8.874,149.551
C08052=1112.417,158.621,-62.830,-179.382,8.871,149.551
C08053=1112.422,158.372,-62.807,-179.384,8.867,149.551
C08054=1112.426,158.122,-62.785,-179.386,8.864,149.551
C08055=1112.431,157.873,-62.762,-179.388,8.861,149.551
C08056=1112.436,157.625,-62.740,-179.391,8.858,149.551
C08057=1112.440,157.376,-62.716,-179.392,8.855,149.550
C08058=1112.445,157.126,-62.694,-179.395,8.851,149.550
C08059=1112.449,156.878,-62.672,-179.397,8.848,149.550
C08060=1112.454,156.629,-62.649,-179.399,8.845,149.550
C08061=1112.458,156.380,-62.627,-179.401,8.841,149.550
C08062=1112.464,156.131,-62.604,-179.404,8.838,149.550
C08063=1112.468,155.882,-62.582,-179.406,8.835,149.549
C08064=1112.472,155.633,-62.560,-179.408,8.831,149.549
C08065=1112.478,155.384,-62.537,-179.410,8.828,149.549
C08066=1112.482,155.135,-62.514,-179.413,8.825,149.549
C08067=1112.486,154.886,-62.492,-179.415,8.821,149.549
C08068=1112.491,154.638,-62.469,-179.416,8.818,149.548
C08069=1112.495,154.388,-62.447,-179.419,8.815,149.548
C08070=1112.500,154.140,-62.426,-179.421,8.812,149.548
C08071=1112.505,153.891,-62.402,-179.423,8.808,149.548
C08072=1112.509,153.641,-62.380,-179.425,8.805,149.548
C08073=1112.514,153.393,-62.359,-179.427,8.802,149.548
C08074=1112.519,153.144,-62.335,-179.429,8.798,149.547
C08075=1112.524,152.895,-62.314,-179.431,8.795,149.547
C08076=1112.528,152.646,-62.292,-179.434,8.791,149.547
C08077=1112.532,152.397,-62.269,-179.436,8.788,149.547
C08078=1112.538,152.148,-62.246,-179.438,8.785,149.547
C08079=1112.542,151.899,-62.224,-179.440,8.781,149.546
C08080=1112.547,151.650,-62.203,-179.442,8.778,149.546
C08081=1112.551,151.401,-62.181,-179.444,8.774,149.546
C08082=1112.556,151.152,-62.158,-179.447,8.771,149.546
C08083=1112.561,150.903,-62.136,-179.449,8.767,149.545
C08084=1112.565,150.654,-62.114,-179.451,8.764,149.545
C08085=1112.570,150.405,-62.092,-179.453,8.760,149.545
C08086=1112.574,150.156,-62.070,-179.455,8.757,149.545
C08087=1112.579,149.907,-62.047,-179.457,8.753,149.545
C08088=1112.583,149.658,-62.025,-179.459,8.750,149.544
C08089=1112.588,149.409,-62.003,-179.461,8.746,149.544
C08090=1112.593,149.160,-61.981,-179.464,8.743,149.544
C08091=1112.597,148.911,-61.959,-179.465,8.739,149.544
C08092=1112.602,148.662,-61.937,-179.468,8.735,149.543
C08093=1112.607,148.413,-61.915,-179.470,8.732,149.543
C08094=1112.612,148.164,-61.893,-179.472,8.728,149.543
C08095=1112.616,147.915,-61.871,-179.474,8.725,149.543
C08096=1112.621,147.666,-61.849,-179.476,8.721,149.542
C08097=1112.626,147.417,-61.828,-179.478,8.718,149.542
C08098=1112.630,147.168,-61.806,-179.480,8.714,149.542
C08099=1112.635,146.919,-61.784,-179.483,8.711,149.542
C08100=1112.639,146.705,-61.765,-179.485,8.707,149.541
C08101=1112.642,146.492,-61.746,-179.486,8.705,149.541
C08102=1112.647,146.278,-61.727,-179.488,8.701,149.541
C08103=1112.651,146.065,-61.709,-179.490,8.698,149.541
C08104=1112.655,145.851,-61.690,-179.492,8.695,149.541
C08105=1112.659,145.637,-61.671,-179.493,8.692,149.540
C08106=1112.663,145.423,-61.652,-179.495,8.689,149.540
C08107=1112.667,145.210,-61.634,-179.497,8.685,149.540
C08108=1112.672,144.961,-61.612,-179.498,8.682,149.539
C08109=1112.676,144.712,-61.590,-179.500,8.679,149.539
C08110=1112.681,144.463,-61.568,-179.502,8.675,149.539
C08111=1112.686,144.214,-61.546,-179.503,8.672,149.538
C08112=1112.690,143.965,-61.525,-179.505,8.668,149.538
C08113=1112.695,143.716,-61.503,-179.507,8.665,149.538
C08114=1112.700,143.467,-61.482,-179.508,8.662,149.537
C08115=1112.703,143.218,-61.460,-179.510,8.658,149.537
C08116=1112.708,142.969,-61.438,-179.512,8.654,149.537
C08117=1112.713,142.720,-61.417,-179.513,8.651,149.536
C08118=1112.717,142.471,-61.395,-179.515,8.648,149.536
C08119=1112.723,142.222,-61.374,-179.517,8.644,149.536
C08120=1112.727,141.973,-61.352,-179.518,8.641,149.536
C08121=1112.732,141.724,-61.330,-179.520,8.638,149.535
C08122=1112.737,141.475,-61.308,-179.522,8.634,149.535
C08123=1112.741,141.225,-61.287,-179.523,8.631,149.534
C08124=1112.746,140.977,-61.265,-179.525,8.627,149.534
C08125=1112.751,140.728,-61.244,-179.527,8.624,149.534
C08126=1112.754,140.479,-61.222,-179.528,8.621,149.534
C08127=1112.760,140.230,-61.201,-179.530,8.617,149.533
C08128=1112.764,139.981,-61.180,-179.532,8.614,149.533
C08129=1112.769,139.732,-61.158,-179.534,8.611,149.533
C08130=1112.774,139.482,-61.137,-179.535,8.607,149.532
C08131=1112.779,139.234,-61.115,-179.537,8.603,149.532
C08132=1112.783,138.985,-61.093,-179.539,8.601,149.532
C08133=1112.788,138.736,-61.072,-179.540,8.597,149.531
C08134=1112.792,138.487,-61.051,-179.542,8.593,149.531
C08135=1112.797,138.237,-61.029,-179.544,8.591,149.531
C08136=1112.802,137.988,-61.008,-179.545,8.587,149.530
C08137=1112.807,137.740,-60.986,-179.548,8.583,149.530
C08138=1112.811,137.490,-60.965,-179.549,8.580,149.530
C08139=1112.815,137.241,-60.944,-179.551,8.577,149.530
C08140=1112.821,136.992,-60.923,-179.553,8.573,149.529
C08141=1112.825,136.743,-60.901,-179.554,8.570,149.529
C08142=1112.830,136.494,-60.880,-179.556,8.567,149.529
C08143=1112.834,136.245,-60.859,-179.558,8.563,149.528
C08144=1112.839,135.996,-60.838,-179.559,8.560,149.528
C08145=1112.844,135.747,-60.816,-179.561,8.557,149.528
C08146=1112.849,135.497,-60.795,-179.563,8.553,149.527
C08147=1112.853,135.249,-60.773,-179.564,8.550,149.527
C08148=1112.858,135.000,-60.753,-179.566,8.546,149.527
C08149=1112.863,134.751,-60.731,-179.568,8.543,149.527
C08150=1112.867,134.501,-60.710,-179.569,8.540,149.526
C08151=1112.872,134.253,-60.688,-179.571,8.536,149.526
C08152=1112.877,134.004,-60.667,-179.573,8.533,149.526
C08153=1112.881,133.755,-60.647,-179.575,8.530,149.525
C08154=1112.886,133.505,-60.625,-179.576,8.526,149.525
C08155=1112.891,133.256,-60.604,-179.578,8.523,149.525
C08156=1112.895,133.043,-60.586,-179.580,8.520,149.525
C08157=1112.899,132.829,-60.569,-179.581,8.517,149.524
C08158=1112.903,132.615,-60.549,-179.583,8.515,149.524
C08159=1112.907,132.402,-60.531,-179.584,8.512,149.524
C08160=1112.911,132.188,-60.514,-179.585,8.509,149.523
C08161=1112.915,131.974,-60.495,-179.587,8.506,149.523
C08162=1112.919,131.760,-60.478,-179.589,8.503,149.523
C08163=1112.923,131.547,-60.459,-179.590,8.500,149.523
C08164=1112.927,131.297,-60.439,-179.592,8.497,149.523
C08165=1112.932,131.048,-60.418,-179.594,8.494,149.522
C08166=1112.937,130.800,-60.397,-179.595,8.490,149.522
C08167=1112.942,130.550,-60.376,-179.597,8.487,149.522
C08168=1112.947,130.301,-60.355,-179.599,8.484,149.521
C08169=1112.951,130.052,-60.334,-179.601,8.480,149.521
C08170=1112.956,129.803,-60.313,-179.602,8.477,149.521
C08171=1112.960,129.554,-60.292,-179.604,8.474,149.521
C08172=1112.965,129.305,-60.271,-179.606,8.470,149.520
C08173=1112.970,129.056,-60.250,-179.607,8.467,149.520
C08174=1112.975,128.807,-60.229,-179.609,8.463,149.520
C08175=1112.979,128.558,-60.208,-179.611,8.460,149.519
C08176=1112.984,128.309,-60.187,-179.613,8.457,149.519
C08177=1112.989,128.059,-60.166,-179.615,8.454,149.519
C08178=1112.994,127.811,-60.146,-179.616,8.450,149.519
C08179=1112.999,127.561,-60.125,-179.618,8.447,149.518
C08180=1113.003,127.312,-60.104,-179.620,8.444,149.518
C08181=1113.008,127.063,-60.083,-179.622,8.440,149.518
C08182=1113.012,126.814,-60.062,-179.623,8.437,149.517
C08183=1113.017,126.565,-60.041,-179.625,8.434,149.517
C08184=1113.022,126.316,-60.021,-179.627,8.430,149.517
C08185=1113.026,126.067,-60.001,-179.629,8.427,149.517
C08186=1113.031,125.818,-59.980,-179.630,8.424,149.516
C08187=1113.036,125.569,-59.959,-179.632,8.420,149.516
C08188=1113.041,125.319,-59.938,-179.634,8.417,149.516
C08189=1113.045,125.070,-59.918,-179.636,8.414,149.516
C08190=1113.051,124.821,-59.897,-179.637,8.410,149.515
C08191=1113.055,124.572,-59.877,-179.639,8.406,149.515
C08192=1113.059,124.323,-59.856,-179.641,8.404,149.515
C08193=1113.065,124.074,-59.835,-179.643,8.400,149.514
C08194=1113.069,123.825,-59.815,-179.644,8.396,149.514
C08195=1113.073,123.575,-59.794,-179.646,8.394,149.514
C08196=1113.078,123.326,-59.773,-179.648,8.390,149.514
C08197=1113.082,123.077,-59.753,-179.650,8.387,149.513
C08198=1113.088,122.828,-59.732,-179.651,8.384,149.513
C08199=1113.092,122.579,-59.711,-179.653,8.380,149.513
C08200=1113.097,122.330,-59.691,-179.655,8.377,149.512
C08201=1113.102,122.081,-59.670,-179.657,8.373,149.512
C08202=1113.106,121.831,-59.650,-179.659,8.370,149.512
C08203=1113.111,121.582,-59.630,-179.660,8.366,149.512
C08204=1113.116,121.333,-59.609,-179.662,8.363,149.511
C08205=1113.121,121.084,-59.589,-179.664,8.360,149.511
C08206=1113.126,120.836,-59.569,-179.666,8.357,149.511
C08207=1113.130,120.587,-59.548,-179.667,8.353,149.510
C08208=1113.135,120.338,-59.527,-179.670,8.349,149.510
C08209=1113.140,120.088,-59.508,-179.671,8.347,149.510
C08210=1113.144,119.839,-59.487,-179.673,8.343,149.510
C08211=1113.149,119.590,-59.467,-179.675,8.339,149.509
C08212=1113.153,119.376,-59.450,-179.676,8.337,149.509
C08213=1113.157,119.162,-59.432,-179.678,8.334,149.509
C08214=1113.161,118.948,-59.414,-179.679,8.331,149.509
C08215=1113.165,118.734,-59.397,-179.680,8.328,149.508
C08216=1113.169,118.521,-59.380,-179.682,8.325,149.508
C08217=1113.174,118.307,-59.362,-179.684,8.322,149.508
C08218=1113.178,118.093,-59.345,-179.685,8.319,149.508
C08219=1113.182,117.879,-59.327,-179.687,8.317,149.508
C08220=1113.187,117.630,-59.307,-179.688,8.313,149.507
C08221=1113.191,117.381,-59.287,-179.690,8.309,149.507
C08222=1113.196,117.132,-59.267,-179.692,8.307,149.507
C08223=1113.200,116.883,-59.247,-179.694,8.303,149.506
C08224=1113.205,116.634,-59.226,-179.696,8.299,149.506
C08225=1113.210,116.384,-59.206,-179.698,8.296,149.506
C08226=1113.215,116.135,-59.186,-179.699,8.293,149.506
C08227=1113.219,115.886,-59.165,-179.701,8.290,149.505
C08228=1113.224,115.637,-59.146,-179.703,8.286,149.505
C08229=1113.229,115.388,-59.126,-179.705,8.282,149.505
C08230=1113.234,115.139,-59.106,-179.706,8.279,149.504
C08231=1113.238,114.890,-59.086,-179.708,8.276,149.504
C08232=1113.243,114.640,-59.065,-179.710,8.272,149.504
C08233=1113.248,114.391,-59.045,-179.712,8.269,149.504
C08234=1113.252,114.142,-59.025,-179.714,8.265,149.503
C08235=1113.258,113.893,-59.005,-179.715,8.262,149.503
C08236=1113.262,113.644,-58.985,-179.717,8.258,149.503
C08237=1113.267,113.395,-58.965,-179.719,8.255,149.502
C08238=1113.271,113.146,-58.945,-179.721,8.251,149.502
C08239=1113.276,112.896,-58.925,-179.722,8.248,149.502
C08240=1113.281,112.648,-58.905,-179.724,8.245,149.502
C08241=1113.286,112.398,-58.886,-179.726,8.241,149.501
C08242=1113.291,112.149,-58.866,-179.728,8.237,149.501
C08243=1113.295,111.900,-58.846,-179.730,8.234,149.501
C08244=1113.300,111.650,-58.826,-179.731,8.231,149.500
C08245=1113.305,111.402,-58.806,-179.733,8.227,149.500
C08246=1113.310,111.152,-58.786,-179.735,8.224,149.500
C08247=1113.315,110.902,-58.766,-179.737,8.220,149.499
C08248=1113.319,110.653,-58.746,-179.739,8.217,149.499
C08249=1113.325,110.405,-58.726,-179.741,8.213,149.499
C08250=1113.328,110.156,-58.707,-179.743,8.210,149.499
C08251=1113.333,109.906,-58.687,-179.745,8.206,149.498
C08252=1113.338,109.657,-58.667,-179.747,8.201,149.498
C08253=1113.343,109.409,-58.647,-179.749,8.198,149.498
C08254=1113.348,109.159,-58.628,-179.751,8.194,149.498
C08255=1113.353,108.909,-58.608,-179.753,8.191,149.497
C08256=1113.357,108.660,-58.588,-179.755,8.187,149.497
C08257=1113.362,108.412,-58.568,-179.757,8.183,149.497
C08258=1113.367,108.162,-58.549,-179.759,8.180,149.496
C08259=1113.372,107.912,-58.529,-179.761,8.176,149.496
C08260=1113.377,107.664,-58.510,-179.763,8.172,149.496
C08261=1113.382,107.415,-58.489,-179.765,8.168,149.496
C08262=1113.386,107.165,-58.470,-179.767,8.164,149.495
C08263=1113.390,106.916,-58.451,-179.769,8.161,149.495
C08264=1113.396,106.667,-58.431,-179.771,8.157,149.495
C08265=1113.400,106.417,-58.412,-179.773,8.154,149.494
C08266=1113.405,106.168,-58.391,-179.775,8.150,149.494
C08267=1113.410,105.920,-58.372,-179.776,8.146,149.494
C08268=1113.414,105.705,-58.356,-179.778,8.143,149.493
C08269=1113.418,105.492,-58.338,-179.780,8.140,149.493
C08270=1113.422,105.278,-58.322,-179.782,8.136,149.493
C08271=1113.426,105.064,-58.305,-179.783,8.133,149.492
C08272=1113.430,104.850,-58.289,-179.785,8.130,149.492
C08273=1113.434,104.636,-58.271,-179.786,8.127,149.492
C08274=1113.438,104.422,-58.255,-179.788,8.123,149.492
C08275=1113.443,104.207,-58.239,-179.789,8.120,149.491
C08276=1113.448,103.959,-58.219,-179.791,8.117,149.491
C08277=1113.452,103.710,-58.200,-179.793,8.113,149.491
C08278=1113.457,103.460,-58.180,-179.795,8.109,149.490
C08279=1113.462,103.211,-58.161,-179.796,8.105,149.490
C08280=1113.467,102.962,-58.141,-179.798,8.102,149.490
C08281=1113.471,102.713,-58.122,-179.800,8.098,149.489
C08282=1113.476,102.464,-58.103,-179.802,8.094,149.489
C08283=1113.481,102.214,-58.083,-179.804,8.090,149.489
C08284=1113.486,101.965,-58.064,-179.806,8.086,149.488
C08285=1113.490,101.715,-58.045,-179.807,8.082,149.488
C08286=1113.496,101.467,-58.026,-179.810,8.078,149.487
C08287=1113.500,101.217,-58.006,-179.811,8.075,149.487
C08288=1113.505,100.968,-57.988,-179.813,8.071,149.487
C08289=1113.510,100.719,-57.968,-179.815,8.067,149.486
C08290=1113.515,100.469,-57.948,-179.816,8.063,149.486
C08291=1113.519,100.221,-57.930,-179.818,8.059,149.485
C08292=1113.524,99.971,-57.910,-179.820,8.056,149.485
C08293=1113.529,99.722,-57.891,-179.821,8.052,149.485
C08294=1113.534,99.472,-57.872,-179.823,8.048,149.484
C08295=1113.539,99.224,-57.853,-179.825,8.044,149.484
C08296=1113.543,98.974,-57.834,-179.826,8.041,149.484
C08297=1113.548,98.726,-57.815,-179.827,8.037,149.483
C08298=1113.553,98.476,-57.795,-179.829,8.033,149.483
C08299=1113.558,98.227,-57.777,-179.831,8.029,149.482
C08300=1113.563,97.977,-57.757,-179.832,8.026,149.482
C08301=1113.567,97.729,-57.739,-179.834,8.022,149.481
C08302=1113.572,97.479,-57.719,-179.835,8.018,149.481
C08303=1113.577,97.231,-57.700,-179.838,8.014,149.481
C08304=1113.582,96.980,-57.681,-179.839,8.010,149.480
C08305=1113.587,96.731,-57.662,-179.841,8.007,149.480
C08306=1113.591,96.482,-57.643,-179.842,8.003,149.479
C08307=1113.597,96.233,-57.624,-179.844,7.999,149.479
C08308=1113.601,95.983,-57.605,-179.846,7.995,149.479
C08309=1113.606,95.735,-57.586,-179.847,7.991,149.478
C08310=1113.611,95.485,-57.568,-179.849,7.987,149.478
C08311=1113.616,95.236,-57.548,-179.850,7.984,149.477
C08312=1113.620,94.987,-57.530,-179.851,7.980,149.477
C08313=1113.625,94.737,-57.511,-179.853,7.976,149.476
C08314=1113.630,94.489,-57.492,-179.854,7.972,149.476
C08315=1113.635,94.239,-57.472,-179.856,7.968,149.475
C08316=1113.640,93.990,-57.455,-179.857,7.964,149.475
C08317=1113.644,93.741,-57.436,-179.859,7.960,149.474
C08318=1113.649,93.491,-57.417,-179.860,7.956,149.474
C08319=1113.654,93.242,-57.398,-179.861,7.953,149.474
C08320=1113.659,92.992,-57.379,-179.863,7.949,149.473
C08321=1113.663,92.744,-57.361,-179.865,7.945,149.473
C08322=1113.669,92.494,-57.342,-179.866,7.942,149.472
C08323=1113.673,92.245,-57.323,-179.867,7.937,149.472
C08324=1113.677,92.031,-57.307,-179.869,7.935,149.471
C08325=1113.681,91.818,-57.291,-179.870,7.931,149.471
C08326=1113.686,91.603,-57.274,-179.871,7.928,149.471
C08327=1113.690,91.389,-57.258,-179.872,7.924,149.470
C08328=1113.694,91.175,-57.242,-179.873,7.921,149.470
C08329=1113.698,90.961,-57.227,-179.874,7.918,149.469
C08330=1113.702,90.747,-57.211,-179.876,7.914,149.469
C08331=1113.706,90.533,-57.195,-179.877,7.911,149.468
C08332=1113.711,90.284,-57.176,-179.878,7.907,149.468
C08333=1113.716,90.035,-57.158,-179.880,7.903,149.467
C08334=1113.721,89.785,-57.139,-179.881,7.900,149.467
C08335=1113.726,89.536,-57.120,-179.882,7.896,149.466
C08336=1113.731,89.287,-57.102,-179.884,7.892,149.466
C08337=1113.735,89.037,-57.083,-179.885,7.888,149.466
C08338=1113.740,88.788,-57.064,-179.886,7.885,149.465
C08339=1113.745,88.539,-57.046,-179.887,7.881,149.464
C08340=1113.749,88.290,-57.027,-179.889,7.877,149.464
C08341=1113.755,88.040,-57.009,-179.891,7.873,149.464
C08342=1113.760,87.791,-56.991,-179.891,7.870,149.463
C08343=1113.764,87.542,-56.972,-179.893,7.866,149.463
C08344=1113.769,87.292,-56.954,-179.894,7.862,149.462
C08345=1113.774,87.043,-56.935,-179.895,7.858,149.461
C08346=1113.778,86.794,-56.916,-179.896,7.854,149.461
C08347=1113.783,86.545,-56.898,-179.898,7.851,149.461
C08348=1113.788,86.295,-56.880,-179.899,7.846,149.460
C08349=1113.794,86.046,-56.862,-179.900,7.843,149.460
C08350=1113.798,85.797,-56.843,-179.901,7.839,149.459
C08351=1113.803,85.547,-56.825,-179.903,7.835,149.458
C08352=1113.808,85.298,-56.807,-179.904,7.832,149.458
C08353=1113.813,85.049,-56.788,-179.905,7.828,149.457
C08354=1113.817,84.800,-56.769,-179.906,7.824,149.457
C08355=1113.822,84.550,-56.751,-179.907,7.820,149.456
C08356=1113.827,84.301,-56.733,-179.909,7.816,149.456
C08357=1113.832,84.052,-56.715,-179.910,7.812,149.455
C08358=1113.836,83.802,-56.697,-179.911,7.809,149.455
C08359=1113.842,83.553,-56.677,-179.912,7.805,149.454
C08360=1113.847,83.304,-56.659,-179.913,7.802,149.454
C08361=1113.852,83.055,-56.641,-179.914,7.798,149.453
C08362=1113.856,82.805,-56.623,-179.915,7.793,149.453
C08363=1113.861,82.556,-56.605,-179.916,7.790,149.452
C08364=1113.866,82.307,-56.587,-179.918,7.786,149.452
C08365=1113.871,82.057,-56.569,-179.919,7.783,149.451
C08366=1113.876,81.808,-56.551,-179.920,7.779,149.450
C08367=1113.881,81.558,-56.532,-179.921,7.775,149.450
C08368=1113.885,81.310,-56.514,-179.922,7.771,149.449
C08369=1113.890,81.060,-56.496,-179.923,7.767,149.449
C08370=1113.895,80.811,-56.478,-179.924,7.764,149.448
C08371=1113.900,80.562,-56.460,-179.925,7.760,149.448
C08372=1113.905,80.313,-56.442,-179.926,7.756,149.447
C08373=1113.909,80.063,-56.423,-179.928,7.753,149.447
C08374=1113.914,79.814,-56.405,-179.928,7.749,149.446
C08375=1113.919,79.565,-56.387,-179.930,7.745,149.446
C08376=1113.924,79.315,-56.369,-179.930,7.742,149.445
C08377=1113.929,79.066,-56.351,-179.932,7.738,149.445
C08378=1113.934,78.817,-56.333,-179.932,7.734,149.444
C08379=1113.939,78.568,-56.315,-179.933,7.730,149.443
C08380=1113.943,78.353,-56.300,-179.934,7.727,149.443
C08381=1113.947,78.139,-56.284,-179.935,7.724,149.442
C08382=1113.951,77.925,-56.269,-179.936,7.721,149.442
C08383=1113.956,77.710,-56.254,-179.937,7.718,149.442
C08384=1113.960,77.497,-56.238,-179.938,7.714,149.441
C08385=1113.964,77.282,-56.222,-179.939,7.711,149.441
C08386=1113.968,77.069,-56.207,-179.940,7.708,149.440
C08387=1113.972,76.854,-56.192,-179.941,7.705,149.440
C08388=1113.977,76.605,-56.174,-179.942,7.700,149.439
C08389=1113.982,76.356,-56.156,-179.943,7.696,149.439
C08390=1113.987,76.107,-56.138,-179.944,7.693,149.438
C08391=1113.992,75.857,-56.121,-179.946,7.689,149.438
C08392=1113.997,75.608,-56.103,-179.947,7.685,149.437
C08393=1114.001,75.358,-56.084,-179.948,7.681,149.437
C08394=1114.006,75.109,-56.066,-179.950,7.677,149.436
C08395=1114.011,74.860,-56.048,-179.952,7.673,149.436
C08396=1114.016,74.611,-56.030,-179.953,7.669,149.435
C08397=1114.021,74.361,-56.013,-179.954,7.665,149.435
C08398=1114.026,74.112,-55.995,-179.956,7.661,149.434
C08399=1114.031,73.862,-55.977,-179.957,7.657,149.434
C08400=1114.036,73.613,-55.959,-179.959,7.653,149.433
C08401=1114.040,73.364,-55.942,-179.960,7.649,149.433
C08402=1114.045,73.115,-55.925,-179.962,7.645,149.432
C08403=1114.050,72.865,-55.907,-179.962,7.642,149.432
C08404=1114.055,72.616,-55.889,-179.964,7.638,149.431
C08405=1114.060,72.366,-55.871,-179.965,7.634,149.431
C08406=1114.065,72.117,-55.853,-179.967,7.630,149.430
C08407=1114.070,71.868,-55.835,-179.968,7.626,149.430
C08408=1114.074,71.619,-55.818,-179.970,7.622,149.429
C08409=1114.079,71.369,-55.801,-179.971,7.618,149.429
C08410=1114.084,71.120,-55.783,-179.972,7.614,149.428
C08411=1114.090,70.870,-55.765,-179.974,7.610,149.428
C08412=1114.094,70.621,-55.747,-179.976,7.606,149.427
C08413=1114.099,70.372,-55.730,-179.977,7.602,149.427
C08414=1114.104,70.123,-55.713,-179.978,7.598,149.426
C08415=1114.109,69.873,-55.695,-179.979,7.595,149.426
C08416=1114.114,69.624,-55.677,-179.980,7.590,149.425
C08417=1114.119,69.374,-55.660,-179.982,7.587,149.425
C08418=1114.123,69.126,-55.642,-179.983,7.583,149.424
C08419=1114.128,68.876,-55.625,-179.985,7.578,149.424
C08420=1114.133,68.627,-55.607,-179.986,7.574,149.423
C08421=1114.138,68.377,-55.590,-179.988,7.571,149.423
C08422=1114.143,68.128,-55.572,-179.989,7.566,149.422
C08423=1114.148,67.878,-55.555,-179.990,7.562,149.422
C08424=1114.153,67.629,-55.537,-179.992,7.558,149.421
C08425=1114.157,67.380,-55.520,-179.992,7.555,149.421
C08426=1114.162,67.130,-55.502,-179.994,7.551,149.420
C08427=1114.168,66.881,-55.486,-179.996,7.547,149.420
C08428=1114.172,66.632,-55.468,-179.997,7.543,149.419
C08429=1114.177,66.383,-55.451,-179.998,7.539,149.419
C08430=1114.182,66.133,-55.433,-180.000,7.535,149.418
C08431=1114.187,65.884,-55.416,179.999,7.531,149.418
C08432=1114.192,65.635,-55.398,179.998,7.527,149.417
C08433=1114.197,65.385,-55.381,179.996,7.523,149.417
C08434=1114.201,65.135,-55.364,179.995,7.519,149.416
C08435=1114.206,64.886,-55.346,179.994,7.516,149.416
C08436=1114.210,64.673,-55.332,179.992,7.512,149.415
C08437=1114.215,64.459,-55.317,179.991,7.508,149.415
C08438=1114.219,64.243,-55.302,179.990,7.505,149.414
C08439=1114.223,64.030,-55.288,179.989,7.501,149.414
C08440=1114.227,63.815,-55.272,179.988,7.498,149.413
C08441=1114.231,63.601,-55.258,179.987,7.495,149.413
C08442=1114.236,63.387,-55.243,179.986,7.491,149.412
C08443=1114.240,63.173,-55.228,179.985,7.488,149.412
C08444=1114.245,62.923,-55.211,179.983,7.484,149.412
C08445=1114.250,62.674,-55.195,179.982,7.480,149.411
C08446=1114.255,62.425,-55.177,179.981,7.476,149.410
C08447=1114.259,62.175,-55.160,179.980,7.473,149.410
C08448=1114.264,61.926,-55.143,179.979,7.468,149.409
C08449=1114.270,61.676,-55.125,179.977,7.464,149.409
C08450=1114.274,61.427,-55.108,179.976,7.460,149.408
C08451=1114.280,61.178,-55.091,179.974,7.456,149.408
C08452=1114.284,60.928,-55.075,179.973,7.452,149.407
C08453=1114.289,60.679,-55.057,179.972,7.448,149.407
C08454=1114.294,60.430,-55.040,179.970,7.444,149.406
C08455=1114.299,60.181,-55.023,179.970,7.441,149.406
C08456=1114.304,59.931,-55.006,179.968,7.437,149.405
C08457=1114.309,59.681,-54.989,179.967,7.432,149.405
C08458=1114.314,59.432,-54.972,179.966,7.428,149.404
C08459=1114.318,59.182,-54.956,179.964,7.424,149.404
C08460=1114.324,58.934,-54.938,179.963,7.420,149.403
C08461=1114.328,58.684,-54.921,179.962,7.416,149.402
C08462=1114.333,58.435,-54.904,179.961,7.413,149.402
C08463=1114.338,58.185,-54.887,179.960,7.409,149.401
C08464=1114.344,57.936,-54.871,179.958,7.405,149.401
C08465=1114.348,57.687,-54.854,179.957,7.401,149.401
C08466=1114.353,57.437,-54.837,179.956,7.396,149.400
C08467=1114.358,57.187,-54.820,179.954,7.393,149.399
C08468=1114.363,56.939,-54.804,179.953,7.388,149.399
C08469=1114.368,56.689,-54.786,179.952,7.385,149.398
C08470=1114.372,56.439,-54.770,179.951,7.381,149.398
C08471=1114.378,56.190,-54.753,179.949,7.377,149.397
C08472=1114.383,55.941,-54.736,179.948,7.373,149.397
C08473=1114.387,55.691,-54.720,179.947,7.368,149.396
C08474=1114.392,55.441,-54.702,179.946,7.364,149.396
C08475=1114.398,55.193,-54.686,179.944,7.360,149.395
C08476=1114.402,54.943,-54.669,179.943,7.357,149.394
C08477=1114.407,54.693,-54.652,179.942,7.353,149.394
C08478=1114.412,54.445,-54.636,179.941,7.349,149.393
C08479=1114.417,54.195,-54.619,179.940,7.344,149.393
C08480=1114.422,53.945,-54.602,179.938,7.341,149.392
C08481=1114.427,53.697,-54.585,179.937,7.336,149.392
C08482=1114.432,53.447,-54.569,179.936,7.332,149.391
C08483=1114.437,53.197,-54.552,179.935,7.329,149.391
C08484=1114.442,52.948,-54.535,179.934,7.325,149.390
C08485=1114.446,52.699,-54.519,179.932,7.321,149.389
C08486=1114.452,52.450,-54.503,179.931,7.316,149.389
C08487=1114.457,52.200,-54.486,179.930,7.312,149.388
C08488=1114.461,51.950,-54.469,179.929,7.308,149.388
C08489=1114.467,51.701,-54.453,179.927,7.304,149.387
C08490=1114.471,51.452,-54.436,179.927,7.301,149.387
C08491=1114.476,51.202,-54.419,179.926,7.296,149.386
C08492=1114.481,50.988,-54.405,179.924,7.292,149.386
C08493=1114.485,50.774,-54.391,179.923,7.289,149.385
C08494=1114.489,50.560,-54.377,179.922,7.286,149.385
C08495=1114.494,50.345,-54.363,179.922,7.283,149.384
C08496=1114.498,50.130,-54.349,179.920,7.279,149.384
C08497=1114.502,49.916,-54.334,179.919,7.276,149.383
C08498=1114.506,49.702,-54.320,179.918,7.273,149.383
C08499=1114.510,49.488,-54.307,179.917,7.268,149.382
C08500=1114.515,49.238,-54.289,179.916,7.264,149.382
C08501=1114.520,48.989,-54.273,179.915,7.261,149.381
C08502=1114.525,48.740,-54.257,179.914,7.257,149.380
C08503=1114.530,48.490,-54.241,179.913,7.253,149.380
C08504=1114.535,48.241,-54.224,179.911,7.248,149.379
C08505=1114.540,47.992,-54.208,179.910,7.244,149.379
C08506=1114.545,47.742,-54.192,179.909,7.240,149.378
C08507=1114.550,47.492,-54.175,179.908,7.237,149.378
C08508=1114.555,47.243,-54.158,179.907,7.232,149.377
C08509=1114.560,46.993,-54.142,179.906,7.228,149.376
C08510=1114.565,46.745,-54.126,179.905,7.224,149.376
C08511=1114.569,46.495,-54.110,179.904,7.220,149.375
C08512=1114.575,46.246,-54.094,179.902,7.216,149.375
C08513=1114.579,45.996,-54.077,179.902,7.212,149.374
C08514=1114.585,45.747,-54.062,179.900,7.208,149.373
C08515=1114.589,45.497,-54.045,179.899,7.204,149.373
C08516=1114.594,45.248,-54.029,179.898,7.200,149.372
C08517=1114.599,44.998,-54.013,179.897,7.196,149.372
C08518=1114.605,44.749,-53.996,179.896,7.191,149.371
C08519=1114.609,44.499,-53.980,179.894,7.187,149.371
C08520=1114.615,44.250,-53.964,179.894,7.184,149.370
C08521=1114.619,44.000,-53.948,179.893,7.179,149.369
C08522=1114.624,43.752,-53.931,179.892,7.175,149.369
C08523=1114.629,43.501,-53.915,179.890,7.171,149.368
C08524=1114.634,43.253,-53.899,179.889,7.167,149.368
C08525=1114.639,43.003,-53.883,179.888,7.163,149.367
C08526=1114.644,42.754,-53.867,179.887,7.159,149.366
C08527=1114.649,42.504,-53.851,179.886,7.155,149.366
C08528=1114.654,42.254,-53.835,179.885,7.151,149.365
C08529=1114.659,42.005,-53.819,179.884,7.147,149.365
C08530=1114.664,41.755,-53.803,179.883,7.142,149.364
C08531=1114.669,41.507,-53.787,179.882,7.138,149.363
C08532=1114.673,41.257,-53.771,179.881,7.134,149.363
C08533=1114.678,41.008,-53.755,179.880,7.131,149.362
C08534=1114.683,40.758,-53.739,179.878,7.126,149.362
C08535=1114.689,40.508,-53.724,179.877,7.122,149.361
C08536=1114.694,40.260,-53.707,179.876,7.118,149.360
C08537=1114.698,40.010,-53.691,179.875,7.113,149.360
C08538=1114.704,39.760,-53.676,179.874,7.109,149.359
C08539=1114.708,39.511,-53.659,179.874,7.106,149.358
C08540=1114.714,39.261,-53.643,179.872,7.102,149.358
C08541=1114.719,39.012,-53.628,179.871,7.097,149.357
C08542=1114.724,38.762,-53.611,179.870,7.093,149.357
C08543=1114.729,38.513,-53.596,179.869,7.089,149.356
C08544=1114.733,38.263,-53.580,179.868,7.084,149.355
C08545=1114.738,38.014,-53.565,179.867,7.081,149.355
C08546=1114.743,37.765,-53.548,179.866,7.077,149.354
C08547=1114.748,37.515,-53.532,179.865,7.072,149.353
C08548=1114.753,37.301,-53.519,179.864,7.069,149.353
C08549=1114.757,37.086,-53.505,179.863,7.065,149.352
C08550=1114.761,36.872,-53.491,179.862,7.062,149.352
C08551=1114.766,36.657,-53.478,179.862,7.058,149.351
C08552=1114.770,36.443,-53.465,179.860,7.054,149.351
C08553=1114.774,36.228,-53.451,179.860,7.051,149.350
C08554=1114.778,36.014,-53.438,179.859,7.048,149.350
C08555=1114.782,35.800,-53.424,179.858,7.043,149.349
C08556=1114.788,35.551,-53.408,179.858,7.040,149.348
C08557=1114.793,35.301,-53.393,179.856,7.035,149.348
C08558=1114.798,35.052,-53.377,179.855,7.031,149.347
C08559=1114.803,34.802,-53.361,179.854,7.027,149.346
C08560=1114.807,34.553,-53.346,179.853,7.023,149.346
C08561=1114.813,34.304,-53.330,179.852,7.018,149.345
C08562=1114.818,34.054,-53.314,179.851,7.014,149.344
C08563=1114.823,33.804,-53.298,179.851,7.010,149.344
C08564=1114.828,33.555,-53.283,179.850,7.006,149.343
C08565=1114.833,33.306,-53.268,179.849,7.002,149.342
C08566=1114.838,33.056,-53.252,179.848,6.997,149.342
C08567=1114.843,32.807,-53.237,179.846,6.993,149.341
C08568=1114.848,32.557,-53.221,179.845,6.989,149.340
C08569=1114.853,32.307,-53.205,179.845,6.985,149.340
C08570=1114.858,32.058,-53.190,179.844,6.981,149.339
C08571=1114.863,31.809,-53.175,179.843,6.977,149.338
C08572=1114.868,31.559,-53.159,179.842,6.972,149.338
C08573=1114.873,31.309,-53.143,179.841,6.968,149.337
C08574=1114.878,31.060,-53.128,179.840,6.964,149.336
C08575=1114.883,30.811,-53.113,179.839,6.959,149.336
C08576=1114.888,30.561,-53.097,179.838,6.956,149.335
C08577=1114.892,30.311,-53.082,179.838,6.951,149.334
C08578=1114.898,30.062,-53.066,179.836,6.947,149.334
C08579=1114.902,29.813,-53.051,179.835,6.943,149.333
C08580=1114.908,29.564,-53.036,179.834,6.938,149.332
C08581=1114.913,29.314,-53.020,179.833,6.934,149.332
C08582=1114.917,29.064,-53.005,179.832,6.930,149.331
C08583=1114.923,28.815,-52.989,179.832,6.926,149.330
C08584=1114.928,28.566,-52.973,179.831,6.922,149.330
C08585=1114.933,28.316,-52.958,179.830,6.917,149.329
C08586=1114.938,28.067,-52.943,179.829,6.913,149.328
C08587=1114.942,27.817,-52.928,179.828,6.908,149.328
C08588=1114.948,27.567,-52.913,179.827,6.904,149.327
C08589=1114.952,27.318,-52.898,179.826,6.900,149.326
C08590=1114.958,27.069,-52.882,179.826,6.896,149.325
C08591=1114.963,26.819,-52.866,179.825,6.892,149.325
C08592=1114.968,26.570,-52.851,179.824,6.887,149.324
C08593=1114.973,26.320,-52.836,179.823,6.883,149.323
C08594=1114.978,26.070,-52.821,179.822,6.879,149.323
C08595=1114.983,25.821,-52.806,179.821,6.874,149.322
C08596=1114.988,25.572,-52.791,179.820,6.870,149.321
C08597=1114.993,25.323,-52.775,179.819,6.865,149.321
C08598=1114.998,25.073,-52.761,179.819,6.862,149.320
C08599=1115.003,24.823,-52.745,179.818,6.857,149.319
C08600=1115.008,24.574,-52.730,179.817,6.853,149.318
C08601=1115.013,24.324,-52.715,179.816,6.849,149.318
C08602=1115.018,24.075,-52.700,179.815,6.844,149.317
C08603=1115.023,23.825,-52.684,179.814,6.840,149.316
C08604=1115.027,23.610,-52.672,179.814,6.836,149.316
C08605=1115.032,23.397,-52.659,179.814,6.832,149.315
C08606=1115.036,23.182,-52.646,179.812,6.829,149.314
C08607=1115.040,22.967,-52.633,179.812,6.825,149.314
C08608=1115.045,22.753,-52.620,179.811,6.821,149.313
C08609=1115.049,22.538,-52.607,179.810,6.817,149.312
C08610=1115.053,22.323,-52.594,179.810,6.814,149.312
C08611=1115.058,22.110,-52.581,179.809,6.810,149.311
C08612=1115.063,21.860,-52.567,179.808,6.806,149.311
C08613=1115.067,21.610,-52.551,179.808,6.801,149.310
C08614=1115.072,21.361,-52.536,179.807,6.797,149.309
C08615=1115.077,21.111,-52.521,179.806,6.792,149.308
C08616=1115.083,20.862,-52.506,179.805,6.788,149.307
C08617=1115.088,20.612,-52.491,179.804,6.783,149.307
C08618=1115.092,20.363,-52.476,179.803,6.779,149.306
C08619=1115.098,20.113,-52.462,179.802,6.774,149.305
C08620=1115.103,19.864,-52.447,179.802,6.771,149.305
C08621=1115.107,19.615,-52.432,179.801,6.766,149.304
C08622=1115.113,19.365,-52.417,179.800,6.762,149.303
C08623=1115.118,19.116,-52.402,179.800,6.757,149.302
C08624=1115.123,18.866,-52.387,179.799,6.753,149.302
C08625=1115.128,18.616,-52.372,179.798,6.748,149.301
C08626=1115.133,18.367,-52.358,179.797,6.744,149.300
C08627=1115.138,18.118,-52.343,179.796,6.739,149.299
C08628=1115.143,17.868,-52.328,179.795,6.735,149.298
C08629=1115.148,17.619,-52.313,179.795,6.730,149.298
C08630=1115.153,17.369,-52.298,179.794,6.727,149.297
C08631=1115.158,17.119,-52.283,179.794,6.722,149.296
C08632=1115.163,16.870,-52.269,179.793,6.718,149.295
C08633=1115.168,16.620,-52.254,179.792,6.713,149.294
C08634=1115.173,16.371,-52.239,179.791,6.708,149.294
C08635=1115.179,16.121,-52.224,179.791,6.704,149.293
C08636=1115.183,15.872,-52.209,179.790,6.699,149.292
C08637=1115.188,15.622,-52.195,179.789,6.695,149.291
C08638=1115.193,15.372,-52.181,179.789,6.690,149.291
C08639=1115.199,15.123,-52.165,179.788,6.686,149.290
C08640=1115.203,14.873,-52.151,179.788,6.682,149.289
C08641=1115.208,14.624,-52.137,179.787,6.677,149.288
C08642=1115.213,14.375,-52.122,179.786,6.673,149.287
C08643=1115.219,14.125,-52.108,179.785,6.668,149.287
C08644=1115.224,13.875,-52.093,179.784,6.664,149.286
C08645=1115.229,13.626,-52.078,179.784,6.659,149.285
C08646=1115.234,13.377,-52.064,179.783,6.654,149.284
C08647=1115.239,13.127,-52.049,179.782,6.650,149.284
C08648=1115.244,12.878,-52.034,179.782,6.645,149.283
C08649=1115.249,12.628,-52.020,179.781,6.641,149.282
C08650=1115.254,12.378,-52.005,179.780,6.636,149.281
C08651=1115.259,12.128,-51.991,179.780,6.632,149.280
C08652=1115.264,11.879,-51.976,179.779,6.627,149.279
C08653=1115.269,11.630,-51.962,179.779,6.623,149.279
C08654=1115.274,11.381,-51.948,179.778,6.619,149.278
C08655=1115.279,11.131,-51.934,179.777,6.614,149.277
C08656=1115.284,10.882,-51.919,179.777,6.609,149.276
C08657=1115.290,10.632,-51.904,179.776,6.605,149.275
C08658=1115.295,10.382,-51.889,179.775,6.600,149.274
C08659=1115.299,10.132,-51.875,179.775,6.595,149.274
C08660=1115.304,9.918,-51.863,179.774,6.592,149.273
C08661=1115.308,9.704,-51.851,179.773,6.588,149.272
C08662=1115.312,9.489,-51.838,179.773,6.584,149.271
C08663=1115.317,9.275,-51.826,179.772,6.579,149.271
C08664=1115.321,9.060,-51.814,179.772,6.576,149.270
C08665=1115.326,8.845,-51.801,179.772,6.572,149.269
C08666=1115.330,8.631,-51.789,179.771,6.568,149.269
C08667=1115.334,8.416,-51.777,179.771,6.564,149.268
C08668=1115.340,8.131,-51.760,179.770,6.558,149.267
C08669=1115.345,7.846,-51.744,179.769,6.553,149.266
C08670=1115.350,7.596,-51.730,179.769,6.549,149.265
C08671=1115.356,7.346,-51.715,179.768,6.544,149.264
C08672=1115.362,7.097,-51.701,179.768,6.539,149.263
C08673=1115.367,6.847,-51.687,179.767,6.535,149.263
C08674=1115.372,6.598,-51.672,179.766,6.530,149.262
C08675=1115.377,6.348,-51.658,179.766,6.526,149.261
C08676=1115.382,6.098,-51.644,179.766,6.522,149.260
C08677=1115.386,5.850,-51.630,179.765,6.517,149.259
C08678=1115.391,5.600,-51.616,179.765,6.512,149.258
C08679=1115.396,5.350,-51.602,179.764,6.508,149.257
C08680=1115.401,5.100,-51.588,179.763,6.503,149.257
C08681=1115.407,4.851,-51.574,179.763,6.498,149.256
C08682=1115.412,4.602,-51.559,179.762,6.494,149.255
C08683=1115.417,4.352,-51.545,179.761,6.489,149.254
C08684=1115.422,4.102,-51.531,179.760,6.485,149.253
C08685=1115.427,3.853,-51.517,179.761,6.481,149.252
C08686=1115.432,3.604,-51.503,179.760,6.476,149.252
C08687=1115.437,3.354,-51.488,179.759,6.471,149.251
C08688=1115.442,3.104,-51.474,179.758,6.467,149.250
C08689=1115.448,2.855,-51.460,179.758,6.462,149.249
C08690=1115.453,2.605,-51.446,179.757,6.458,149.248
C08691=1115.458,2.355,-51.432,179.757,6.453,149.247
C08692=1115.462,2.106,-51.419,179.756,6.448,149.246
C08693=1115.468,1.857,-51.405,179.755,6.444,149.246
C08694=1115.473,1.607,-51.390,179.755,6.440,149.245
C08695=1115.477,1.357,-51.376,179.755,6.435,149.244
C08696=1115.483,1.108,-51.362,179.754,6.430,149.243
C08697=1115.488,0.859,-51.348,179.753,6.426,149.242
C08698=1115.493,0.608,-51.334,179.753,6.421,149.242
C08699=1115.497,0.359,-51.321,179.752,6.417,149.241
C08700=1115.503,0.110,-51.307,179.751,6.412,149.240
C08701=1115.508,-0.140,-51.293,179.751,6.408,149.239
C08702=1115.513,-0.390,-51.278,179.751,6.404,149.238
C08703=1115.519,-0.639,-51.265,179.750,6.399,149.237
C08704=1115.524,-0.889,-51.251,179.749,6.395,149.237
C08705=1115.528,-1.138,-51.237,179.749,6.390,149.236
C08706=1115.534,-1.387,-51.223,179.748,6.385,149.235
C08707=1115.539,-1.638,-51.210,179.748,6.381,149.234
C08708=1115.544,-1.887,-51.195,179.747,6.376,149.233
C08709=1115.549,-2.136,-51.182,179.746,6.371,149.232
C08710=1115.554,-2.386,-51.169,179.746,6.367,149.232
C08711=1115.559,-2.635,-51.155,179.745,6.363,149.231
C08712=1115.564,-2.885,-51.140,179.745,6.358,149.230
C08713=1115.569,-3.135,-51.126,179.744,6.354,149.229
C08714=1115.574,-3.384,-51.113,179.743,6.349,149.228
C08715=1115.579,-3.634,-51.099,179.743,6.345,149.228
C08716=1115.584,-3.884,-51.085,179.742,6.340,149.227
C08717=1115.589,-4.133,-51.072,179.742,6.335,149.226
C08718=1115.596,-4.419,-51.056,179.741,6.331,149.225
C08719=1115.601,-4.707,-51.040,179.740,6.325,149.224
C08720=1115.607,-4.993,-51.025,179.740,6.320,149.223
C08721=1115.613,-5.280,-51.010,179.739,6.314,149.222
C08722=1115.618,-5.529,-50.995,179.738,6.310,149.221
C08723=1115.623,-5.780,-50.982,179.737,6.305,149.220
C08724=1115.628,-6.028,-50.968,179.737,6.301,149.220
C08725=1115.633,-6.278,-50.954,179.736,6.297,149.219
C08726=1115.639,-6.528,-50.941,179.736,6.292,149.218
C08727=1115.643,-6.777,-50.927,179.735,6.288,149.217
C08728=1115.649,-7.027,-50.914,179.735,6.283,149.216
C08729=1115.654,-7.277,-50.900,179.734,6.279,149.216
C08730=1115.659,-7.526,-50.887,179.733,6.274,149.215
C08731=1115.664,-7.776,-50.873,179.733,6.269,149.214
C08732=1115.669,-8.025,-50.860,179.732,6.265,149.213
C08733=1115.674,-8.275,-50.846,179.731,6.260,149.212
C08734=1115.680,-8.525,-50.832,179.731,6.255,149.211
C08735=1115.684,-8.774,-50.819,179.731,6.252,149.211
C08736=1115.690,-9.024,-50.806,179.730,6.247,149.210
C08737=1115.694,-9.273,-50.792,179.729,6.242,149.209
C08738=1115.700,-9.523,-50.779,179.729,6.238,149.208
C08739=1115.705,-9.772,-50.766,179.728,6.233,149.207
C08740=1115.710,-10.022,-50.752,179.727,6.229,149.206
C08741=1115.716,-10.272,-50.739,179.727,6.224,149.206
C08742=1115.720,-10.521,-50.725,179.726,6.220,149.205
C08743=1115.726,-10.771,-50.712,179.725,6.215,149.204
C08744=1115.730,-11.021,-50.699,179.725,6.210,149.203
C08745=1115.736,-11.270,-50.685,179.724,6.205,149.202
C08746=1115.740,-11.520,-50.672,179.723,6.201,149.202
C08747=1115.746,-11.769,-50.659,179.723,6.196,149.201
C08748=1115.750,-12.019,-50.645,179.722,6.192,149.200
C08749=1115.756,-12.268,-50.632,179.722,6.187,149.199
C08750=1115.761,-12.518,-50.619,179.722,6.183,149.198
C08751=1115.766,-12.767,-50.605,179.721,6.179,149.197
C08752=1115.771,-13.017,-50.592,179.721,6.174,149.196
C08753=1115.777,-13.267,-50.579,179.720,6.169,149.196
C08754=1115.782,-13.516,-50.565,179.719,6.165,149.195
C08755=1115.787,-13.766,-50.552,179.719,6.160,149.194
C08756=1115.792,-14.015,-50.539,179.718,6.155,149.193
C08757=1115.797,-14.266,-50.526,179.718,6.151,149.192
C08758=1115.802,-14.514,-50.512,179.717,6.146,149.192
C08759=1115.807,-14.764,-50.500,179.716,6.142,149.191
C08760=1115.812,-15.014,-50.486,179.716,6.137,149.190
C08761=1115.817,-15.263,-50.474,179.715,6.132,149.189
C08762=1115.822,-15.513,-50.459,179.714,6.128,149.188
C08763=1115.828,-15.762,-50.447,179.714,6.123,149.187
C08764=1115.833,-16.012,-50.434,179.713,6.118,149.186
C08765=1115.838,-16.262,-50.421,179.713,6.114,149.185
C08766=1115.843,-16.511,-50.408,179.712,6.109,149.185
C08767=1115.848,-16.762,-50.394,179.711,6.104,149.184
C08768=1115.853,-17.010,-50.381,179.711,6.100,149.183
C08769=1115.858,-17.260,-50.369,179.710,6.095,149.182
C08770=1115.862,-17.475,-50.357,179.710,6.091,149.181
C08771=1115.867,-17.690,-50.346,179.709,6.087,149.181
C08772=1115.872,-17.904,-50.334,179.709,6.083,149.180
C08773=1115.876,-18.120,-50.324,179.708,6.079,149.179
C08774=1115.880,-18.334,-50.313,179.708,6.075,149.179
C08775=1115.885,-18.549,-50.301,179.707,6.071,149.178
C08776=1115.889,-18.763,-50.290,179.707,6.067,149.177
C08777=1115.893,-18.978,-50.279,179.706,6.063,149.176
C08778=1115.899,-19.228,-50.266,179.705,6.058,149.175
C08779=1115.904,-19.477,-50.253,179.705,6.053,149.175
C08780=1115.909,-19.727,-50.240,179.704,6.048,149.174
C08781=1115.914,-19.977,-50.227,179.704,6.044,149.173
C08782=1115.920,-20.226,-50.214,179.703,6.039,149.172
C08783=1115.924,-20.476,-50.201,179.703,6.034,149.171
C08784=1115.930,-20.726,-50.189,179.702,6.030,149.170
C08785=1115.935,-20.975,-50.175,179.702,6.025,149.169
C08786=1115.940,-21.225,-50.163,179.701,6.020,149.168
C08787=1115.945,-21.474,-50.150,179.701,6.016,149.168
C08788=1115.950,-21.724,-50.137,179.700,6.011,149.167
C08789=1115.956,-21.973,-50.124,179.700,6.006,149.166
C08790=1115.961,-22.223,-50.111,179.699,6.002,149.165
C08791=1115.966,-22.473,-50.099,179.699,5.997,149.164
C08792=1115.971,-22.722,-50.086,179.698,5.992,149.163
C08793=1115.977,-22.972,-50.073,179.698,5.987,149.162
C08794=1115.981,-23.222,-50.060,179.697,5.983,149.161
C08795=1115.986,-23.471,-50.047,179.697,5.978,149.160
C08796=1115.992,-23.721,-50.035,179.696,5.972,149.159
C08797=1115.997,-23.970,-50.023,179.695,5.968,149.159
C08798=1116.002,-24.221,-50.009,179.695,5.963,149.158
C08799=1116.007,-24.470,-49.997,179.694,5.958,149.157
C08800=1116.012,-24.719,-49.984,179.694,5.953,149.156
C08801=1116.018,-24.969,-49.971,179.693,5.949,149.155
C08802=1116.022,-25.219,-49.958,179.693,5.944,149.154
C08803=1116.028,-25.469,-49.946,179.692,5.939,149.153
C08804=1116.033,-25.718,-49.934,179.692,5.934,149.152
C08805=1116.039,-25.967,-49.921,179.691,5.930,149.151
C08806=1116.044,-26.217,-49.908,179.692,5.925,149.150
C08807=1116.048,-26.467,-49.895,179.693,5.921,149.149
C08808=1116.054,-26.717,-49.883,179.693,5.917,149.148
C08809=1116.059,-26.966,-49.871,179.693,5.913,149.147
C08810=1116.064,-27.215,-49.858,179.694,5.909,149.146
C08811=1116.069,-27.465,-49.845,179.694,5.905,149.145
C08812=1116.074,-27.715,-49.833,179.695,5.900,149.144
C08813=1116.079,-27.965,-49.821,179.694,5.896,149.143
C08814=1116.085,-28.214,-49.807,179.694,5.892,149.142
C08815=1116.090,-28.464,-49.795,179.695,5.887,149.141
C08816=1116.095,-28.714,-49.783,179.695,5.883,149.140
C08817=1116.100,-28.964,-49.770,179.695,5.878,149.139
C08818=1116.105,-29.213,-49.757,179.695,5.874,149.138
C08819=1116.110,-29.462,-49.745,179.695,5.870,149.137
C08820=1116.116,-29.712,-49.733,179.696,5.866,149.136
C08821=1116.121,-29.961,-49.720,179.696,5.861,149.135
C08822=1116.126,-30.211,-49.708,179.696,5.857,149.134
C08823=1116.131,-30.461,-49.695,179.695,5.853,149.133
C08824=1116.136,-30.711,-49.683,179.695,5.849,149.132
C08825=1116.141,-30.960,-49.670,179.696,5.845,149.131
C08826=1116.146,-31.175,-49.660,179.696,5.841,149.131
C08827=1116.150,-31.389,-49.649,179.695,5.837,149.130
C08828=1116.155,-31.605,-49.638,179.695,5.833,149.129
C08829=1116.158,-31.820,-49.627,179.695,5.830,149.128
C08830=1116.164,-32.035,-49.617,179.695,5.826,149.128
C08831=1116.168,-32.249,-49.606,179.694,5.821,149.127
C08832=1116.172,-32.464,-49.596,179.694,5.818,149.126
C08833=1116.177,-32.679,-49.585,179.694,5.814,149.125
C08834=1116.182,-32.928,-49.573,179.694,5.810,149.124
C08835=1116.187,-33.178,-49.560,179.693,5.806,149.124
C08836=1116.193,-33.428,-49.548,179.693,5.801,149.123
C08837=1116.197,-33.678,-49.535,179.692,5.796,149.122
C08838=1116.203,-33.928,-49.523,179.693,5.792,149.121
C08839=1116.208,-34.177,-49.511,179.692,5.787,149.120
C08840=1116.213,-34.427,-49.499,179.692,5.783,149.119
C08841=1116.218,-34.676,-49.486,179.691,5.778,149.118
C08842=1116.223,-34.925,-49.474,179.690,5.774,149.117
C08843=1116.229,-35.175,-49.462,179.690,5.770,149.117
C08844=1116.233,-35.424,-49.450,179.690,5.765,149.116
C08845=1116.239,-35.674,-49.438,179.689,5.761,149.115
C08846=1116.244,-35.924,-49.425,179.689,5.756,149.114
C08847=1116.249,-36.174,-49.413,179.688,5.751,149.113
C08848=1116.254,-36.423,-49.401,179.688,5.746,149.112
C08849=1116.260,-36.673,-49.389,179.686,5.741,149.112
C08850=1116.265,-36.923,-49.377,179.686,5.737,149.111
C08851=1116.270,-37.173,-49.364,179.685,5.732,149.110
C08852=1116.275,-37.423,-49.352,179.684,5.727,149.109
C08853=1116.280,-37.672,-49.340,179.684,5.723,149.108
C08854=1116.285,-37.922,-49.328,179.683,5.717,149.107
C08855=1116.290,-38.171,-49.316,179.682,5.713,149.107
C08856=1116.296,-38.421,-49.304,179.681,5.708,149.106
C08857=1116.301,-38.671,-49.292,179.680,5.702,149.105
C08858=1116.306,-38.920,-49.279,179.679,5.698,149.104
C08859=1116.311,-39.170,-49.267,179.679,5.693,149.103
C08860=1116.316,-39.420,-49.256,179.678,5.688,149.102
C08861=1116.321,-39.669,-49.244,179.677,5.683,149.102
C08862=1116.327,-39.919,-49.232,179.676,5.678,149.101
C08863=1116.332,-40.169,-49.220,179.676,5.673,149.100
C08864=1116.337,-40.418,-49.207,179.674,5.668,149.099
C08865=1116.343,-40.667,-49.196,179.673,5.663,149.098
C08866=1116.348,-40.917,-49.184,179.673,5.658,149.097
C08867=1116.353,-41.166,-49.172,179.671,5.653,149.097
C08868=1116.359,-41.416,-49.160,179.670,5.647,149.096
C08869=1116.363,-41.666,-49.149,179.669,5.642,149.095
C08870=1116.369,-41.916,-49.137,179.668,5.636,149.094
C08871=1116.374,-42.165,-49.124,179.667,5.632,149.093
C08872=1116.379,-42.415,-49.112,179.666,5.626,149.092
C08873=1116.384,-42.665,-49.101,179.665,5.621,149.091
C08874=1116.389,-42.915,-49.089,179.664,5.615,149.091
C08875=1116.395,-43.165,-49.077,179.663,5.610,149.090
C08876=1116.399,-43.414,-49.065,179.664,5.605,149.089
C08877=1116.405,-43.664,-49.053,179.664,5.601,149.087
C08878=1116.410,-43.914,-49.041,179.664,5.596,149.086
C08879=1116.415,-44.162,-49.030,179.664,5.591,149.085
C08880=1116.421,-44.412,-49.019,179.664,5.587,149.084
C08881=1116.426,-44.662,-49.007,179.665,5.581,149.083
C08882=1116.431,-44.877,-48.997,179.665,5.577,149.082
C08883=1116.435,-45.092,-48.987,179.665,5.574,149.081
C08884=1116.439,-45.307,-48.977,179.665,5.570,149.080
C08885=1116.444,-45.522,-48.967,179.665,5.566,149.079
C08886=1116.449,-45.737,-48.956,179.665,5.562,149.078
C08887=1116.453,-45.952,-48.946,179.666,5.558,149.078
C08888=1116.457,-46.167,-48.936,179.666,5.554,149.077
C08889=1116.462,-46.382,-48.926,179.665,5.549,149.076
C08890=1116.467,-46.632,-48.914,179.666,5.545,149.075
C08891=1116.472,-46.881,-48.903,179.666,5.540,149.073
C08892=1116.477,-47.131,-48.891,179.666,5.536,149.073
C08893=1116.482,-47.380,-48.880,179.666,5.531,149.071
C08894=1116.488,-47.630,-48.868,179.666,5.525,149.070
C08895=1116.493,-47.880,-48.856,179.667,5.521,149.069
C08896=1116.498,-48.130,-48.845,179.667,5.516,149.068
C08897=1116.503,-48.379,-48.833,179.667,5.512,149.067
C08898=1116.508,-48.629,-48.822,179.667,5.507,149.066
C08899=1116.514,-48.878,-48.810,179.667,5.502,149.065
C08900=1116.520,-49.128,-48.798,179.668,5.498,149.064
C08901=1116.524,-49.378,-48.787,179.668,5.493,149.063
C08902=1116.530,-49.628,-48.775,179.668,5.489,149.062
C08903=1116.534,-49.877,-48.764,179.668,5.484,149.061
C08904=1116.540,-50.127,-48.752,179.668,5.478,149.059
C08905=1116.545,-50.376,-48.741,179.669,5.474,149.058
C08906=1116.551,-50.626,-48.729,179.668,5.469,149.057
C08907=1116.555,-50.876,-48.718,179.669,5.465,149.056
C08908=1116.561,-51.126,-48.706,179.669,5.460,149.055
C08909=1116.566,-51.375,-48.695,179.669,5.455,149.054
C08910=1116.571,-51.625,-48.683,179.669,5.451,149.053
C08911=1116.576,-51.874,-48.672,179.669,5.446,149.052
C08912=1116.582,-52.124,-48.660,179.670,5.442,149.051
C08913=1116.586,-52.374,-48.649,179.670,5.437,149.050
C08914=1116.593,-52.624,-48.638,179.670,5.431,149.049
C08915=1116.597,-52.873,-48.627,179.670,5.427,149.048
C08916=1116.603,-53.123,-48.615,179.670,5.422,149.047
C08917=1116.607,-53.373,-48.604,179.670,5.417,149.045
C08918=1116.613,-53.622,-48.592,179.670,5.413,149.045
C08919=1116.618,-53.872,-48.581,179.670,5.408,149.043
C08920=1116.624,-54.122,-48.569,179.671,5.404,149.042
C08921=1116.629,-54.372,-48.558,179.671,5.399,149.041
C08922=1116.635,-54.621,-48.547,179.671,5.394,149.040
C08923=1116.639,-54.871,-48.535,179.671,5.390,149.039
C08924=1116.644,-55.120,-48.524,179.671,5.385,149.038
C08925=1116.649,-55.370,-48.512,179.672,5.380,149.037
C08926=1116.655,-55.619,-48.501,179.672,5.375,149.036
C08927=1116.660,-55.870,-48.490,179.671,5.371,149.035
C08928=1116.665,-56.119,-48.479,179.672,5.366,149.034
C08929=1116.670,-56.369,-48.468,179.672,5.361,149.033
C08930=1116.676,-56.618,-48.456,179.672,5.357,149.032
C08931=1116.681,-56.869,-48.446,179.672,5.352,149.030
C08932=1116.686,-57.119,-48.434,179.673,5.347,149.029
C08933=1116.692,-57.367,-48.423,179.673,5.343,149.028
C08934=1116.696,-57.617,-48.411,179.673,5.338,149.027
C08935=1116.702,-57.868,-48.400,179.673,5.334,149.026
C08936=1116.707,-58.117,-48.389,179.673,5.329,149.025
C08937=1116.712,-58.366,-48.378,179.673,5.324,149.024
C08938=1116.716,-58.581,-48.368,179.673,5.320,149.023
C08939=1116.721,-58.797,-48.359,179.674,5.316,149.022
C08940=1116.725,-59.011,-48.349,179.674,5.312,149.021
C08941=1116.730,-59.227,-48.339,179.674,5.308,149.020
C08942=1116.735,-59.441,-48.330,179.674,5.304,149.019
C08943=1116.740,-59.657,-48.321,179.674,5.300,149.019
C08944=1116.744,-59.871,-48.310,179.674,5.296,149.018
C08945=1116.748,-60.086,-48.300,179.674,5.292,149.017
C08946=1116.753,-60.337,-48.290,179.673,5.287,149.016
C08947=1116.758,-60.585,-48.279,179.673,5.282,149.015
C08948=1116.764,-60.836,-48.268,179.672,5.276,149.014
C08949=1116.769,-61.086,-48.257,179.672,5.271,149.013
C08950=1116.774,-61.335,-48.246,179.672,5.267,149.012
C08951=1116.779,-61.585,-48.235,179.671,5.261,149.011
C08952=1116.785,-61.835,-48.223,179.670,5.256,149.010
C08953=1116.790,-62.084,-48.212,179.669,5.251,149.009
C08954=1116.795,-62.334,-48.202,179.669,5.246,149.008
C08955=1116.800,-62.583,-48.191,179.668,5.240,149.007
C08956=1116.806,-62.833,-48.180,179.668,5.235,149.006
C08957=1116.811,-63.083,-48.168,179.668,5.230,149.005
C08958=1116.816,-63.333,-48.158,179.667,5.225,149.004
C08959=1116.821,-63.582,-48.147,179.666,5.220,149.004
C08960=1116.827,-63.832,-48.136,179.666,5.214,149.002
C08961=1116.832,-64.082,-48.125,179.665,5.209,149.001
C08962=1116.837,-64.332,-48.114,179.665,5.205,149.001
C08963=1116.842,-64.581,-48.103,179.665,5.199,148.999
C08964=1116.847,-64.831,-48.093,179.664,5.194,148.998
C08965=1116.853,-65.080,-48.081,179.664,5.189,148.998
C08966=1116.858,-65.331,-48.071,179.663,5.183,148.996
C08967=1116.864,-65.579,-48.060,179.663,5.178,148.995
C08968=1116.869,-65.830,-48.049,179.663,5.173,148.994
C08969=1116.874,-66.080,-48.038,179.662,5.168,148.993
C08970=1116.879,-66.329,-48.028,179.662,5.163,148.992
C08971=1116.884,-66.579,-48.017,179.662,5.158,148.991
C08972=1116.890,-66.828,-48.005,179.661,5.152,148.990
C08973=1116.895,-67.079,-47.995,179.661,5.147,148.989
C08974=1116.900,-67.328,-47.985,179.661,5.142,148.988
C08975=1116.905,-67.578,-47.973,179.660,5.136,148.987
C08976=1116.911,-67.827,-47.963,179.660,5.132,148.986
C08977=1116.916,-68.078,-47.953,179.660,5.127,148.985
C08978=1116.921,-68.326,-47.942,179.659,5.121,148.984
C08979=1116.926,-68.577,-47.931,179.659,5.116,148.983
C08980=1116.932,-68.826,-47.921,179.659,5.111,148.982
C08981=1116.936,-69.076,-47.910,179.658,5.105,148.981
C08982=1116.943,-69.326,-47.899,179.658,5.100,148.980
C08983=1116.948,-69.576,-47.888,179.658,5.095,148.979
C08984=1116.953,-69.825,-47.877,179.658,5.090,148.978
C08985=1116.958,-70.075,-47.867,179.658,5.084,148.976
C08986=1116.964,-70.325,-47.856,179.657,5.079,148.976
C08987=1116.969,-70.574,-47.846,179.657,5.074,148.974
C08988=1116.974,-70.824,-47.835,179.658,5.069,148.973
C08989=1116.979,-71.073,-47.825,179.657,5.063,148.972
C08990=1116.984,-71.324,-47.814,179.657,5.058,148.971
C08991=1116.990,-71.573,-47.804,179.657,5.053,148.970
C08992=1116.995,-71.823,-47.793,179.657,5.048,148.969
C08993=1117.000,-72.072,-47.782,179.657,5.043,148.968
C08994=1117.004,-72.288,-47.774,179.656,5.039,148.967
C08995=1117.009,-72.502,-47.765,179.656,5.034,148.966
C08996=1117.014,-72.718,-47.756,179.656,5.030,148.965
C08997=1117.018,-72.933,-47.747,179.656,5.025,148.964
C08998=1117.023,-73.148,-47.738,179.656,5.020,148.963
C08999=1117.028,-73.363,-47.729,179.656,5.016,148.962
C09000=1117.032,-73.578,-47.720,179.656,5.011,148.961
C09001=1117.037,-73.793,-47.711,179.656,5.007,148.960
C09002=1117.042,-74.043,-47.700,179.656,5.002,148.959
C09003=1117.048,-74.293,-47.690,179.656,4.996,148.958
C09004=1117.053,-74.542,-47.679,179.656,4.991,148.957
C09005=1117.058,-74.792,-47.669,179.656,4.986,148.956
C09006=1117.063,-75.041,-47.659,179.656,4.981,148.955
C09007=1117.068,-75.292,-47.649,179.656,4.976,148.953
C09008=1117.073,-75.541,-47.638,179.656,4.971,148.952
C09009=1117.079,-75.791,-47.628,179.656,4.966,148.951
C09010=1117.084,-76.041,-47.618,179.656,4.960,148.950
C09011=1117.090,-76.291,-47.607,179.656,4.954,148.949
C09012=1117.095,-76.540,-47.597,179.656,4.949,148.948
C09013=1117.100,-76.790,-47.587,179.656,4.944,148.946
C09014=1117.106,-77.040,-47.576,179.656,4.939,148.945
C09015=1117.111,-77.289,-47.567,179.656,4.934,148.944
C09016=1117.116,-77.539,-47.556,179.656,4.929,148.943
C09017=1117.121,-77.789,-47.546,179.656,4.924,148.942
C09018=1117.127,-78.038,-47.536,179.656,4.919,148.941
C09019=1117.132,-78.289,-47.525,179.657,4.914,148.940
C09020=1117.137,-78.538,-47.515,179.657,4.908,148.938
C09021=1117.143,-78.788,-47.505,179.657,4.903,148.937
C09022=1117.148,-79.037,-47.495,179.657,4.898,148.936
C09023=1117.153,-79.287,-47.485,179.657,4.893,148.935
C09024=1117.159,-79.537,-47.474,179.657,4.888,148.934
C09025=1117.164,-79.787,-47.465,179.658,4.883,148.933
C09026=1117.169,-80.037,-47.454,179.658,4.878,148.931
C09027=1117.174,-80.286,-47.445,179.658,4.872,148.930
C09028=1117.180,-80.536,-47.435,179.658,4.867,148.929
C09029=1117.185,-80.786,-47.424,179.659,4.862,148.928
C09030=1117.190,-81.036,-47.414,179.659,4.857,148.927
C09031=1117.195,-81.285,-47.404,179.659,4.851,148.925
C09032=1117.201,-81.535,-47.394,179.659,4.846,148.924
C09033=1117.206,-81.785,-47.383,179.659,4.841,148.923
C09034=1117.212,-82.035,-47.374,179.660,4.836,148.922
C09035=1117.217,-82.284,-47.364,179.660,4.831,148.921
C09036=1117.222,-82.534,-47.354,179.660,4.826,148.919
C09037=1117.227,-82.784,-47.343,179.661,4.821,148.918
C09038=1117.233,-83.033,-47.333,179.661,4.816,148.917
C09039=1117.238,-83.283,-47.324,179.661,4.811,148.916
C09040=1117.244,-83.533,-47.314,179.661,4.806,148.915
C09041=1117.249,-83.783,-47.304,179.662,4.800,148.913
C09042=1117.254,-84.032,-47.294,179.662,4.795,148.912
C09043=1117.259,-84.282,-47.284,179.662,4.790,148.911
C09044=1117.265,-84.532,-47.274,179.663,4.786,148.910
C09045=1117.271,-84.782,-47.264,179.663,4.780,148.909
C09046=1117.275,-85.032,-47.254,179.663,4.775,148.907
C09047=1117.280,-85.281,-47.244,179.663,4.770,148.906
C09048=1117.286,-85.531,-47.234,179.664,4.765,148.905
C09049=1117.291,-85.780,-47.225,179.665,4.760,148.904
C09050=1117.296,-85.996,-47.215,179.665,4.756,148.903
C09051=1117.301,-86.211,-47.208,179.665,4.752,148.902
C09052=1117.305,-86.426,-47.199,179.666,4.747,148.901
C09053=1117.310,-86.641,-47.190,179.666,4.743,148.900
C09054=1117.314,-86.857,-47.182,179.667,4.739,148.899
C09055=1117.319,-87.071,-47.174,179.666,4.734,148.898
C09056=1117.323,-87.287,-47.165,179.667,4.730,148.896
C09057=1117.328,-87.502,-47.157,179.667,4.726,148.895
C09058=1117.333,-87.752,-47.146,179.668,4.721,148.894
C09059=1117.338,-88.001,-47.137,179.668,4.716,148.893
C09060=1117.344,-88.252,-47.127,179.669,4.711,148.892
C09061=1117.349,-88.501,-47.118,179.669,4.706,148.891
C09062=1117.354,-88.750,-47.107,179.670,4.701,148.889
C09063=1117.360,-89.000,-47.098,179.670,4.696,148.888
C09064=1117.364,-89.250,-47.088,179.670,4.691,148.887
C09065=1117.370,-89.501,-47.079,179.671,4.687,148.886
C09066=1117.375,-89.750,-47.069,179.672,4.681,148.884
C09067=1117.381,-89.999,-47.059,179.672,4.676,148.883
C09068=1117.386,-90.249,-47.050,179.673,4.672,148.882
C09069=1117.392,-90.499,-47.040,179.673,4.666,148.881
C09070=1117.397,-90.749,-47.030,179.674,4.662,148.880
C09071=1117.402,-90.999,-47.020,179.674,4.657,148.878
C09072=1117.407,-91.248,-47.010,179.675,4.651,148.877
C09073=1117.412,-91.498,-47.001,179.675,4.647,148.876
C09074=1117.418,-91.748,-46.991,179.676,4.642,148.875
C09075=1117.423,-91.998,-46.982,179.676,4.638,148.873
C09076=1117.429,-92.247,-46.972,179.677,4.632,148.872
C09077=1117.434,-92.497,-46.963,179.678,4.628,148.871
C09078=1117.440,-92.747,-46.953,179.678,4.622,148.870
C09079=1117.444,-92.997,-46.943,179.679,4.618,148.868
C09080=1117.450,-93.247,-46.933,179.679,4.613,148.867
C09081=1117.455,-93.497,-46.924,179.680,4.609,148.866
C09082=1117.461,-93.746,-46.914,179.681,4.604,148.865
C09083=1117.466,-93.996,-46.905,179.681,4.599,148.863
C09084=1117.471,-94.245,-46.895,179.682,4.594,148.862
C09085=1117.476,-94.495,-46.886,179.682,4.589,148.861
C09086=1117.482,-94.745,-46.876,179.683,4.584,148.860
C09087=1117.487,-94.995,-46.867,179.683,4.580,148.859
C09088=1117.493,-95.244,-46.857,179.684,4.575,148.858
C09089=1117.498,-95.494,-46.848,179.684,4.569,148.856
C09090=1117.504,-95.744,-46.838,179.684,4.564,148.855
C09091=1117.508,-95.994,-46.828,179.684,4.560,148.854
C09092=1117.514,-96.244,-46.818,179.684,4.555,148.853
C09093=1117.519,-96.494,-46.809,179.685,4.550,148.852
C09094=1117.524,-96.743,-46.800,179.685,4.545,148.851
C09095=1117.530,-96.993,-46.790,179.686,4.540,148.849
C09096=1117.535,-97.243,-46.781,179.686,4.535,148.848
C09097=1117.540,-97.492,-46.771,179.686,4.530,148.847
C09098=1117.546,-97.742,-46.762,179.686,4.525,148.846
C09099=1117.552,-97.992,-46.753,179.687,4.521,148.845
C09100=1117.556,-98.242,-46.743,179.687,4.515,148.844
C09101=1117.562,-98.491,-46.734,179.688,4.510,148.842
C09102=1117.567,-98.741,-46.724,179.688,4.505,148.841
C09103=1117.572,-98.991,-46.715,179.689,4.501,148.840
C09104=1117.578,-99.241,-46.706,179.689,4.496,148.839
C09105=1117.583,-99.490,-46.696,179.689,4.490,148.838
C09106=1117.588,-99.705,-46.688,179.689,4.486,148.837
C09107=1117.592,-99.921,-46.680,179.689,4.482,148.836
C09108=1117.597,-100.136,-46.673,179.689,4.478,148.835
C09109=1117.602,-100.352,-46.663,179.690,4.473,148.834
C09110=1117.606,-100.567,-46.656,179.690,4.469,148.833
C09111=1117.611,-100.782,-46.648,179.690,4.465,148.832
C09112=1117.615,-100.998,-46.640,179.691,4.460,148.830
C09113=1117.620,-101.212,-46.632,179.691,4.456,148.829
C09114=1117.625,-101.462,-46.623,179.691,4.451,148.828
C09115=1117.631,-101.712,-46.613,179.692,4.446,148.827
C09116=1117.636,-101.962,-46.605,179.692,4.441,148.826
C09117=1117.641,-102.211,-46.595,179.693,4.436,148.825
C09118=1117.647,-102.461,-46.585,179.693,4.431,148.823
C09119=1117.652,-102.711,-46.577,179.693,4.426,148.822
C09120=1117.657,-102.961,-46.568,179.693,4.421,148.821
C09121=1117.663,-103.211,-46.557,179.693,4.416,148.820
C09122=1117.668,-103.461,-46.549,179.693,4.411,148.819
C09123=1117.673,-103.710,-46.540,179.694,4.407,148.818
C09124=1117.678,-103.960,-46.531,179.694,4.402,148.817
C09125=1117.684,-104.210,-46.521,179.695,4.396,148.815
C09126=1117.689,-104.460,-46.512,179.695,4.391,148.814
C09127=1117.694,-104.709,-46.503,179.695,4.386,148.813
C09128=1117.700,-104.959,-46.494,179.695,4.381,148.812
C09129=1117.706,-105.209,-46.485,179.696,4.376,148.811
C09130=1117.711,-105.459,-46.476,179.696,4.371,148.809
C09131=1117.716,-105.708,-46.467,179.697,4.366,148.808
C09132=1117.721,-105.958,-46.457,179.697,4.361,148.807
C09133=1117.727,-106.208,-46.448,179.697,4.356,148.806
C09134=1117.732,-106.458,-46.439,179.697,4.351,148.805
C09135=1117.737,-106.708,-46.430,179.698,4.346,148.803
C09136=1117.743,-106.957,-46.421,179.698,4.340,148.802
C09137=1117.748,-107.207,-46.412,179.698,4.335,148.801
C09138=1117.754,-107.457,-46.403,179.698,4.330,148.800
C09139=1117.759,-107.707,-46.394,179.699,4.325,148.799
C09140=1117.765,-107.956,-46.385,179.699,4.321,148.797
C09141=1117.769,-108.206,-46.376,179.700,4.315,148.796
C09142=1117.775,-108.456,-46.367,179.700,4.310,148.795
C09143=1117.780,-108.706,-46.357,179.700,4.305,148.794
C09144=1117.786,-108.956,-46.348,179.700,4.300,148.793
C09145=1117.791,-109.205,-46.340,179.701,4.295,148.791
C09146=1117.796,-109.455,-46.331,179.701,4.290,148.790
C09147=1117.802,-109.704,-46.322,179.701,4.284,148.789
C09148=1117.807,-109.954,-46.313,179.701,4.279,148.788
C09149=1117.812,-110.204,-46.304,179.702,4.274,148.787
C09150=1117.818,-110.454,-46.295,179.702,4.269,148.785
C09151=1117.823,-110.704,-46.286,179.702,4.264,148.784
C09152=1117.828,-110.954,-46.277,179.702,4.259,148.783
